SPLINE
SPL {X  -136.861, Y  +292.299, Z    +0.000, E1   +47.815, E3 +153540.728}
SPL {X  -156.420, Y  +335.300, Z    +0.000, E1   +31.885, E3 +153548.517}
SPL {X  -161.293, Y  +358.252, Z    +0.000, E1   +18.542, E3 +153550.234}
SPL {X  -162.687, Y  +373.932, Z    +0.000, E1    +7.306, E3 +153550.370}
SPL {X  -162.820, Y  +382.772, Z    +0.000, E1    -0.135, E3 +153549.808}
SPL {X  -162.820, Y  +387.649, Z    +0.000, E1    -8.215, E3 +153549.563}
SPL {X  -162.820, Y  +392.460, Z    +0.000, E1   -17.627, E3 +153549.544}
SPL {X  -162.820, Y  +397.383, Z    +0.000, E1   -27.100, E3 +153549.614}
SPL {X  -162.820, Y  +404.822, Z    +0.000, E1   -40.113, E3 +153549.266}
SPL {X  -162.820, Y  +416.103, Z    +0.000, E1   -54.033, E3 +153549.118}
SPL {X  -162.820, Y  +467.510, Z    +0.000, E1   -69.867, E3 +153562.696}
SPL {X  -162.820, Y  +604.717, Z    +0.000, E1   -70.047, E3 +153644.416}
ENDSPLINE

SPLINE
SPL {X  -162.820, Y  +602.324, Z    +0.000, E1   -67.733, E3 +153661.865}
ENDSPLINE

SPLINE
SPL {X  -162.820, Y  +616.480, Z    +0.000, E1   -67.752, E3 +153673.895}
SPL {X  -162.820, Y  +636.914, Z    +0.000, E1   -67.842, E3 +153690.588}
SPL {X  -162.820, Y  +651.339, Z    +0.000, E1   -67.768, E3 +153703.257}
SPL {X  -162.820, Y  +663.021, Z    +0.000, E1   -67.764, E3 +153713.302}
SPL {X  -162.642, Y  +681.112, Z    +0.000, E1   -67.812, E3 +153728.453}
SPL {X  -161.154, Y  +696.734, Z    +0.000, E1   -67.591, E3 +153743.450}
SPL {X  -159.690, Y  +705.270, Z    +0.000, E1   -67.348, E3 +153752.558}
SPL {X  -157.320, Y  +715.461, Z    +0.000, E1   -67.133, E3 +153763.151}
SPL {X  -154.452, Y  +725.025, Z    +0.000, E1   -66.701, E3 +153774.335}
SPL {X  -152.159, Y  +731.448, Z    +0.000, E1   -66.356, E3 +153782.288}
SPL {X  -148.374, Y  +740.549, Z    +0.000, E1   -65.919, E3 +153793.162}
SPL {X  -144.196, Y  +749.116, Z    +0.000, E1   -65.203, E3 +153804.838}
SPL {X  -141.115, Y  +754.722, Z    +0.000, E1   -64.893, E3 +153811.297}
SPL {X  -138.151, Y  +759.667, Z    +0.000, E1   -64.251, E3 +153819.119}
SPL {X  -134.751, Y  +764.892, Z    +0.000, E1   -63.716, E3 +153826.122}
SPL {X  -131.007, Y  +770.183, Z    +0.000, E1   -63.497, E3 +153831.619}
SPL {X   -85.750, Y  +811.910, Z    +0.000, E1   -55.921, E3 +153935.572}
ENDSPLINE

SPLINE
SPL {X  -114.463, Y  +789.295, Z    +0.000, E1   -54.865, E3 +154104.839}
SPL {X  -149.148, Y  +738.810, Z    +0.000, E1   -41.467, E3 +154115.910}
SPL {X  -159.693, Y  +705.258, Z    +0.000, E1   -25.118, E3 +154118.550}
SPL {X  -162.196, Y  +687.741, Z    +0.000, E1   -13.310, E3 +154119.515}
SPL {X  -162.791, Y  +676.596, Z    +0.000, E1    -4.586, E3 +154119.799}
SPL {X  -162.820, Y  +671.385, Z    +0.000, E1    +0.078, E3 +154119.216}
SPL {X  -162.820, Y  +667.797, Z    +0.000, E1    +5.943, E3 +154118.875}
SPL {X  -162.820, Y  +663.306, Z    +0.000, E1   +14.820, E3 +154118.842}
SPL {X  -162.820, Y  +658.944, Z    +0.000, E1   +23.544, E3 +154119.031}
SPL {X  -162.820, Y  +650.349, Z    +0.000, E1   +39.427, E3 +154118.528}
SPL {X  -162.820, Y  +632.228, Z    +0.000, E1   +60.508, E3 +154117.758}
SPL {X  -162.820, Y  +572.535, Z    +0.000, E1   +70.270, E3 +154139.803}
SPL {X  -162.820, Y  +446.522, Z    +0.000, E1   +69.253, E3 +154223.626}
SPL {X  -162.820, Y  +444.665, Z    +0.000, E1   +68.107, E3 +154235.177}
SPL {X  -162.820, Y  +425.935, Z    +0.000, E1   +68.194, E3 +154250.232}
SPL {X  -162.820, Y  +409.792, Z    +0.000, E1   +68.121, E3 +154264.156}
SPL {X  -162.820, Y  +394.392, Z    +0.000, E1   +68.165, E3 +154276.730}
SPL {X  -162.820, Y  +385.264, Z    +0.000, E1   +67.766, E3 +154287.646}
ENDSPLINE

SPLINE
SPL {X  -162.820, Y  +401.104, Z    +0.000, E1   +65.023, E3 +154295.371}
ENDSPLINE

SPLINE
SPL {X  -162.820, Y  +386.513, Z    +0.000, E1   +65.423, E3 +154306.367}
SPL {X  -161.886, Y  +363.082, Z    +0.000, E1   +66.474, E3 +154319.799}
SPL {X  -158.043, Y  +341.350, Z    +0.000, E1   +67.216, E3 +154332.995}
SPL {X  -154.848, Y  +330.175, Z    +0.000, E1   +66.891, E3 +154344.807}
SPL {X  -151.242, Y  +320.199, Z    +0.000, E1   +66.443, E3 +154356.608}
SPL {X  -147.540, Y  +311.636, Z    +0.000, E1   +65.718, E3 +154368.586}
SPL {X  -144.094, Y  +304.689, Z    +0.000, E1   +65.338, E3 +154376.801}
SPL {X  -141.093, Y  +299.241, Z    +0.000, E1   +65.039, E3 +154383.114}
SPL {X  -138.425, Y  +294.774, Z    +0.000, E1   +64.416, E3 +154390.297}
SPL {X  -135.581, Y  +290.344, Z    +0.000, E1   +63.996, E3 +154396.130}
SPL {X  -132.317, Y  +285.618, Z    +0.000, E1   +63.461, E3 +154402.704}
SPL {X  -126.028, Y  +277.411, Z    +0.000, E1   +65.004, E3 +154402.876}
SPL {X   -85.291, Y  +241.807, Z    +0.000, E1   +53.957, E3 +154549.471}
ENDSPLINE

SPLINE
SPL {X  -136.861, Y  +292.299, Z    +0.000, E1   +47.815, E3 +154677.091}
SPL {X  -156.420, Y  +335.300, Z    +0.000, E1   +31.885, E3 +154684.881}
SPL {X  -161.293, Y  +358.252, Z    +0.000, E1   +18.542, E3 +154686.598}
SPL {X  -162.487, Y  +370.094, Z    +0.000, E1   +10.144, E3 +154686.676}
SPL {X  -162.818, Y  +379.612, Z    +0.000, E1    +2.663, E3 +154686.652}
SPL {X  -162.820, Y  +382.500, Z    +0.000, E1    +0.000, E3 +154686.245}
SPL {X  -162.820, Y  +383.629, Z    +0.000, E1    -1.565, E3 +154685.939}
SPL {X  -162.820, Y  +387.649, Z    +0.000, E1    -8.215, E3 +154685.926}
SPL {X  -162.820, Y  +392.460, Z    +0.000, E1   -17.627, E3 +154685.908}
SPL {X  -162.820, Y  +397.383, Z    +0.000, E1   -27.100, E3 +154685.978}
SPL {X  -162.820, Y  +404.822, Z    +0.000, E1   -40.113, E3 +154685.630}
SPL {X  -162.820, Y  +416.103, Z    +0.000, E1   -54.033, E3 +154685.482}
SPL {X  -162.820, Y  +472.592, Z    +0.000, E1   -70.190, E3 +154701.084}
SPL {X  -162.820, Y  +605.049, Z    +0.000, E1   -68.347, E3 +154795.565}
SPL {X  -162.820, Y  +616.480, Z    +0.000, E1   -67.752, E3 +154810.258}
SPL {X  -162.820, Y  +631.154, Z    +0.000, E1   -67.735, E3 +154822.793}
SPL {X  -162.820, Y  +647.590, Z    +0.000, E1   -67.861, E3 +154835.828}
SPL {X  -162.820, Y  +663.021, Z    +0.000, E1   -67.764, E3 +154849.666}
SPL {X  -162.642, Y  +681.112, Z    +0.000, E1   -67.812, E3 +154864.817}
SPL {X  -161.154, Y  +696.734, Z    +0.000, E1   -67.591, E3 +154879.814}
SPL {X  -158.503, Y  +710.744, Z    +0.000, E1   -67.284, E3 +154894.345}
SPL {X  -155.060, Y  +723.165, Z    +0.000, E1   -66.797, E3 +154908.521}
SPL {X  -151.511, Y  +733.123, Z    +0.000, E1   -66.286, E3 +154920.675}
SPL {X  -147.735, Y  +741.944, Z    +0.000, E1   -65.827, E3 +154931.201}
SPL {X  -144.196, Y  +749.116, Z    +0.000, E1   -65.203, E3 +154941.201}
SPL {X  -139.960, Y  +756.696, Z    +0.000, E1   -64.606, E3 +154951.096}
SPL {X  -135.604, Y  +763.621, Z    +0.000, E1   -63.883, E3 +154960.698}
SPL {X  -131.007, Y  +770.183, Z    +0.000, E1   -63.497, E3 +154967.983}
SPL {X   -85.750, Y  +811.910, Z    +0.000, E1   -55.921, E3 +155071.935}
ENDSPLINE

SPLINE
SPL {X  -114.463, Y  +789.295, Z    +0.000, E1   -54.865, E3 +155241.202}
SPL {X  -149.148, Y  +738.810, Z    +0.000, E1   -41.467, E3 +155252.274}
SPL {X  -159.693, Y  +705.258, Z    +0.000, E1   -25.118, E3 +155254.913}
SPL {X  -162.196, Y  +687.741, Z    +0.000, E1   -13.310, E3 +155255.878}
SPL {X  -162.791, Y  +676.596, Z    +0.000, E1    -4.586, E3 +155256.163}
SPL {X  -162.820, Y  +671.548, Z    +0.000, E1    -0.068, E3 +155255.640}
SPL {X  -162.820, Y  +669.949, Z    +0.000, E1    +2.213, E3 +155255.327}
SPL {X  -162.820, Y  +664.754, Z    +0.000, E1   +11.697, E3 +155255.226}
SPL {X  -162.820, Y  +658.944, Z    +0.000, E1   +23.544, E3 +155255.394}
SPL {X  -162.820, Y  +653.429, Z    +0.000, E1   +34.521, E3 +155254.785}
SPL {X  -162.820, Y  +647.179, Z    +0.000, E1   +44.317, E3 +155255.001}
SPL {X  -162.820, Y  +632.228, Z    +0.000, E1   +60.508, E3 +155254.121}
SPL {X  -162.820, Y  +572.535, Z    +0.000, E1   +70.270, E3 +155276.166}
SPL {X  -162.820, Y  +446.522, Z    +0.000, E1   +69.253, E3 +155359.990}
SPL {X  -162.820, Y  +444.665, Z    +0.000, E1   +68.107, E3 +155371.540}
SPL {X  -162.820, Y  +425.935, Z    +0.000, E1   +68.194, E3 +155386.596}
SPL {X  -162.820, Y  +405.187, Z    +0.000, E1   +68.161, E3 +155404.184}
SPL {X  -162.820, Y  +387.680, Z    +0.000, E1   +67.977, E3 +155420.373}
ENDSPLINE

SPLINE
SPL {X  -162.820, Y  +397.358, Z    +0.000, E1   +65.083, E3 +155435.011}
ENDSPLINE

SPLINE
SPL {X  -162.719, Y  +374.774, Z    +0.000, E1   +65.968, E3 +155449.496}
SPL {X  -160.017, Y  +350.416, Z    +0.000, E1   +67.091, E3 +155462.401}
SPL {X  -156.713, Y  +336.324, Z    +0.000, E1   +67.030, E3 +155474.998}
SPL {X  -153.279, Y  +325.584, Z    +0.000, E1   +66.662, E3 +155486.763}
SPL {X  -149.546, Y  +316.107, Z    +0.000, E1   +66.216, E3 +155497.938}
SPL {X  -147.033, Y  +310.560, Z    +0.000, E1   +65.497, E3 +155507.153}
SPL {X  -144.094, Y  +304.689, Z    +0.000, E1   +65.338, E3 +155513.164}
SPL {X  -141.093, Y  +299.241, Z    +0.000, E1   +65.039, E3 +155519.477}
SPL {X  -138.425, Y  +294.774, Z    +0.000, E1   +64.416, E3 +155526.661}
SPL {X  -134.374, Y  +288.555, Z    +0.000, E1   +63.758, E3 +155535.303}
SPL {X  -128.896, Y  +281.020, Z    +0.000, E1   +64.005, E3 +155540.426}
SPL {X   -85.291, Y  +241.807, Z    +0.000, E1   +53.957, E3 +155685.834}
ENDSPLINE

SPLINE
SPL {X  -136.861, Y  +292.299, Z    +0.000, E1   +47.815, E3 +155813.455}
SPL {X  -156.420, Y  +335.300, Z    +0.000, E1   +31.885, E3 +155821.244}
SPL {X  -161.293, Y  +358.252, Z    +0.000, E1   +18.542, E3 +155822.962}
SPL {X  -162.487, Y  +370.094, Z    +0.000, E1   +10.144, E3 +155823.040}
SPL {X  -162.818, Y  +379.612, Z    +0.000, E1    +2.663, E3 +155823.015}
SPL {X  -162.820, Y  +382.500, Z    +0.000, E1    +0.000, E3 +155822.609}
SPL {X  -162.820, Y  +383.629, Z    +0.000, E1    -1.565, E3 +155822.302}
SPL {X  -162.820, Y  +387.649, Z    +0.000, E1    -8.215, E3 +155822.290}
SPL {X  -162.820, Y  +392.460, Z    +0.000, E1   -17.627, E3 +155822.271}
SPL {X  -162.820, Y  +397.383, Z    +0.000, E1   -27.100, E3 +155822.342}
SPL {X  -162.820, Y  +404.822, Z    +0.000, E1   -40.113, E3 +155821.993}
SPL {X  -162.820, Y  +416.103, Z    +0.000, E1   -54.033, E3 +155821.845}
SPL {X  -162.820, Y  +467.510, Z    +0.000, E1   -69.867, E3 +155835.423}
SPL {X  -162.820, Y  +604.717, Z    +0.000, E1   -70.047, E3 +155917.143}
ENDSPLINE

SPLINE
SPL {X  -162.820, Y  +602.324, Z    +0.000, E1   -67.733, E3 +155934.592}
ENDSPLINE

SPLINE
SPL {X  -162.820, Y  +616.480, Z    +0.000, E1   -67.752, E3 +155946.622}
SPL {X  -162.820, Y  +636.914, Z    +0.000, E1   -67.842, E3 +155963.316}
SPL {X  -162.820, Y  +654.663, Z    +0.000, E1   -67.744, E3 +155979.142}
SPL {X  -162.820, Y  +673.210, Z    +0.000, E1   -67.837, E3 +155994.175}
SPL {X  -162.071, Y  +689.103, Z    +0.000, E1   -67.763, E3 +156008.240}
SPL {X  -160.373, Y  +701.624, Z    +0.000, E1   -67.439, E3 +156021.599}
SPL {X  -157.887, Y  +713.277, Z    +0.000, E1   -67.197, E3 +156033.370}
SPL {X  -155.060, Y  +723.165, Z    +0.000, E1   -66.797, E3 +156044.885}
SPL {X  -151.511, Y  +733.123, Z    +0.000, E1   -66.286, E3 +156057.039}
SPL {X  -148.440, Y  +740.403, Z    +0.000, E1   -65.944, E3 +156065.399}
SPL {X  -146.076, Y  +745.418, Z    +0.000, E1   -65.453, E3 +156072.874}
SPL {X  -142.207, Y  +752.793, Z    +0.000, E1   -65.028, E3 +156081.723}
SPL {X  -139.223, Y  +757.923, Z    +0.000, E1   -64.359, E3 +156089.693}
SPL {X  -135.604, Y  +763.621, Z    +0.000, E1   -63.883, E3 +156097.061}
SPL {X  -131.007, Y  +770.183, Z    +0.000, E1   -63.497, E3 +156104.346}
SPL {X   -85.750, Y  +811.910, Z    +0.000, E1   -55.921, E3 +156208.299}
ENDSPLINE

SPLINE
SPL {X  -114.463, Y  +789.295, Z    +0.000, E1   -54.865, E3 +156377.566}
SPL {X  -144.553, Y  +748.431, Z    +0.000, E1   -44.979, E3 +156388.274}
SPL {X  -156.024, Y  +720.050, Z    +0.000, E1   -33.178, E3 +156389.841}
SPL {X  -160.714, Y  +699.606, Z    +0.000, E1   -21.520, E3 +156391.715}
SPL {X  -162.196, Y  +687.741, Z    +0.000, E1   -13.310, E3 +156392.242}
SPL {X  -162.718, Y  +679.252, Z    +0.000, E1    -6.705, E3 +156392.579}
SPL {X  -162.820, Y  +671.587, Z    +0.000, E1    -0.252, E3 +156391.978}
SPL {X  -162.820, Y  +667.797, Z    +0.000, E1    +5.943, E3 +156391.602}
SPL {X  -162.820, Y  +663.306, Z    +0.000, E1   +14.820, E3 +156391.569}
SPL {X  -162.820, Y  +658.944, Z    +0.000, E1   +23.544, E3 +156391.758}
SPL {X  -162.820, Y  +650.349, Z    +0.000, E1   +39.427, E3 +156391.255}
SPL {X  -162.820, Y  +635.494, Z    +0.000, E1   +57.613, E3 +156390.958}
SPL {X  -162.820, Y  +626.637, Z    +0.000, E1   +64.941, E3 +156389.674}
SPL {X  -162.820, Y  +572.535, Z    +0.000, E1   +70.270, E3 +156412.530}
SPL {X  -162.820, Y  +446.522, Z    +0.000, E1   +69.253, E3 +156496.354}
SPL {X  -162.820, Y  +444.665, Z    +0.000, E1   +68.107, E3 +156507.904}
SPL {X  -162.820, Y  +425.935, Z    +0.000, E1   +68.194, E3 +156522.960}
SPL {X  -162.820, Y  +409.792, Z    +0.000, E1   +68.121, E3 +156536.883}
SPL {X  -162.820, Y  +394.392, Z    +0.000, E1   +68.165, E3 +156549.458}
SPL {X  -162.820, Y  +385.264, Z    +0.000, E1   +67.766, E3 +156560.373}
ENDSPLINE

SPLINE
SPL {X  -162.820, Y  +401.104, Z    +0.000, E1   +65.023, E3 +156568.098}
ENDSPLINE

SPLINE
SPL {X  -162.820, Y  +386.513, Z    +0.000, E1   +65.423, E3 +156579.094}
SPL {X  -162.431, Y  +369.249, Z    +0.000, E1   +66.195, E3 +156589.095}
SPL {X  -160.017, Y  +350.416, Z    +0.000, E1   +67.091, E3 +156598.765}
SPL {X  -156.713, Y  +336.324, Z    +0.000, E1   +67.030, E3 +156611.361}
SPL {X  -153.279, Y  +325.584, Z    +0.000, E1   +66.662, E3 +156623.126}
SPL {X  -149.546, Y  +316.107, Z    +0.000, E1   +66.216, E3 +156634.302}
SPL {X  -147.033, Y  +310.560, Z    +0.000, E1   +65.497, E3 +156643.516}
SPL {X  -144.094, Y  +304.689, Z    +0.000, E1   +65.338, E3 +156649.528}
SPL {X  -141.093, Y  +299.241, Z    +0.000, E1   +65.039, E3 +156655.841}
SPL {X  -138.425, Y  +294.774, Z    +0.000, E1   +64.416, E3 +156663.025}
SPL {X  -135.581, Y  +290.344, Z    +0.000, E1   +63.996, E3 +156668.857}
SPL {X  -133.378, Y  +287.116, Z    +0.000, E1   +63.482, E3 +156674.021}
SPL {X  -128.896, Y  +281.020, Z    +0.000, E1   +64.005, E3 +156676.790}
SPL {X   -85.291, Y  +241.807, Z    +0.000, E1   +53.957, E3 +156822.198}
ENDSPLINE

SPLINE
SPL {X  -136.861, Y  +292.299, Z    +0.000, E1   +47.815, E3 +156949.819}
SPL {X  -156.420, Y  +335.300, Z    +0.000, E1   +31.885, E3 +156957.608}
SPL {X  -161.293, Y  +358.252, Z    +0.000, E1   +18.542, E3 +156959.325}
SPL {X  -162.487, Y  +370.094, Z    +0.000, E1   +10.144, E3 +156959.404}
SPL {X  -162.818, Y  +379.612, Z    +0.000, E1    +2.663, E3 +156959.379}
SPL {X  -162.820, Y  +382.928, Z    +0.000, E1    -0.395, E3 +156958.856}
SPL {X  -162.820, Y  +386.448, Z    +0.000, E1    -6.246, E3 +156958.611}
SPL {X  -162.820, Y  +391.031, Z    +0.000, E1   -14.627, E3 +156958.670}
SPL {X  -162.820, Y  +397.383, Z    +0.000, E1   -27.100, E3 +156958.705}
SPL {X  -162.820, Y  +404.822, Z    +0.000, E1   -40.113, E3 +156958.357}
SPL {X  -162.820, Y  +416.103, Z    +0.000, E1   -54.033, E3 +156958.209}
SPL {X  -162.820, Y  +467.510, Z    +0.000, E1   -69.867, E3 +156971.787}
SPL {X  -162.820, Y  +604.717, Z    +0.000, E1   -70.047, E3 +157053.507}
SPL {X  -162.820, Y  +606.663, Z    +0.000, E1   -67.762, E3 +157074.555}
SPL {X  -162.820, Y  +620.455, Z    +0.000, E1   -67.717, E3 +157086.528}
SPL {X  -162.820, Y  +636.914, Z    +0.000, E1   -67.842, E3 +157099.679}
SPL {X  -162.820, Y  +654.663, Z    +0.000, E1   -67.744, E3 +157115.505}
SPL {X  -162.820, Y  +673.210, Z    +0.000, E1   -67.837, E3 +157130.539}
SPL {X  -162.071, Y  +689.103, Z    +0.000, E1   -67.763, E3 +157144.604}
SPL {X  -160.908, Y  +698.381, Z    +0.000, E1   -67.466, E3 +157154.843}
SPL {X  -159.690, Y  +705.270, Z    +0.000, E1   -67.348, E3 +157161.648}
SPL {X  -157.320, Y  +715.461, Z    +0.000, E1   -67.133, E3 +157172.242}
SPL {X  -154.452, Y  +725.025, Z    +0.000, E1   -66.701, E3 +157183.426}
SPL {X  -151.511, Y  +733.123, Z    +0.000, E1   -66.286, E3 +157193.402}
SPL {X  -147.735, Y  +741.944, Z    +0.000, E1   -65.827, E3 +157203.928}
SPL {X  -144.196, Y  +749.116, Z    +0.000, E1   -65.203, E3 +157213.929}
SPL {X  -139.960, Y  +756.696, Z    +0.000, E1   -64.606, E3 +157223.823}
SPL {X  -136.860, Y  +761.702, Z    +0.000, E1   -64.057, E3 +157230.817}
SPL {X  -134.751, Y  +764.892, Z    +0.000, E1   -63.716, E3 +157235.212}
SPL {X  -131.007, Y  +770.183, Z    +0.000, E1   -63.497, E3 +157240.710}
SPL {X   -85.750, Y  +811.910, Z    +0.000, E1   -55.921, E3 +157344.663}
ENDSPLINE

SPLINE
SPL {X  -114.463, Y  +789.295, Z    +0.000, E1   -54.865, E3 +157513.930}
SPL {X  -149.148, Y  +738.810, Z    +0.000, E1   -41.467, E3 +157525.001}
SPL {X  -159.693, Y  +705.258, Z    +0.000, E1   -25.118, E3 +157527.640}
SPL {X  -162.196, Y  +687.741, Z    +0.000, E1   -13.310, E3 +157528.606}
SPL {X  -162.718, Y  +679.252, Z    +0.000, E1    -6.705, E3 +157528.943}
SPL {X  -162.820, Y  +671.809, Z    +0.000, E1    -0.439, E3 +157528.409}
SPL {X  -162.820, Y  +669.949, Z    +0.000, E1    +2.213, E3 +157528.054}
SPL {X  -162.820, Y  +664.754, Z    +0.000, E1   +11.697, E3 +157527.953}
SPL {X  -162.820, Y  +658.944, Z    +0.000, E1   +23.544, E3 +157528.122}
SPL {X  -162.820, Y  +650.349, Z    +0.000, E1   +39.427, E3 +157527.619}
SPL {X  -162.820, Y  +632.228, Z    +0.000, E1   +60.508, E3 +157526.849}
SPL {X  -162.820, Y  +572.535, Z    +0.000, E1   +70.270, E3 +157548.893}
SPL {X  -162.820, Y  +446.522, Z    +0.000, E1   +69.253, E3 +157632.717}
SPL {X  -162.820, Y  +444.665, Z    +0.000, E1   +68.107, E3 +157644.267}
SPL {X  -162.820, Y  +425.935, Z    +0.000, E1   +68.194, E3 +157659.323}
SPL {X  -162.820, Y  +405.187, Z    +0.000, E1   +68.161, E3 +157676.912}
SPL {X  -162.820, Y  +387.680, Z    +0.000, E1   +67.977, E3 +157693.100}
ENDSPLINE

SPLINE
SPL {X  -162.820, Y  +397.358, Z    +0.000, E1   +65.083, E3 +157707.739}
ENDSPLINE

SPLINE
SPL {X  -162.719, Y  +374.774, Z    +0.000, E1   +65.968, E3 +157722.223}
SPL {X  -160.017, Y  +350.416, Z    +0.000, E1   +67.091, E3 +157735.129}
SPL {X  -156.713, Y  +336.324, Z    +0.000, E1   +67.030, E3 +157747.725}
SPL {X  -153.279, Y  +325.584, Z    +0.000, E1   +66.662, E3 +157759.490}
SPL {X  -150.291, Y  +317.867, Z    +0.000, E1   +66.312, E3 +157768.409}
SPL {X  -147.540, Y  +311.636, Z    +0.000, E1   +65.718, E3 +157777.677}
SPL {X  -144.094, Y  +304.689, Z    +0.000, E1   +65.338, E3 +157785.892}
SPL {X  -141.093, Y  +299.241, Z    +0.000, E1   +65.039, E3 +157792.204}
SPL {X  -138.425, Y  +294.774, Z    +0.000, E1   +64.416, E3 +157799.388}
SPL {X  -134.374, Y  +288.555, Z    +0.000, E1   +63.758, E3 +157808.031}
SPL {X  -128.896, Y  +281.020, Z    +0.000, E1   +64.005, E3 +157813.153}
SPL {X   -85.291, Y  +241.807, Z    +0.000, E1   +53.957, E3 +157958.561}
ENDSPLINE

SPLINE
SPL {X  -136.861, Y  +292.299, Z    +0.000, E1   +47.815, E3 +158086.182}
SPL {X  -156.420, Y  +335.300, Z    +0.000, E1   +31.885, E3 +158093.972}
SPL {X  -161.293, Y  +358.252, Z    +0.000, E1   +18.542, E3 +158095.689}
SPL {X  -162.487, Y  +370.094, Z    +0.000, E1   +10.144, E3 +158095.767}
SPL {X  -162.818, Y  +379.612, Z    +0.000, E1    +2.663, E3 +158095.743}
SPL {X  -162.820, Y  +382.928, Z    +0.000, E1    -0.395, E3 +158095.220}
SPL {X  -162.820, Y  +387.649, Z    +0.000, E1    -8.215, E3 +158095.017}
SPL {X  -162.820, Y  +392.460, Z    +0.000, E1   -17.627, E3 +158094.999}
SPL {X  -162.820, Y  +397.383, Z    +0.000, E1   -27.100, E3 +158095.069}
SPL {X  -162.820, Y  +404.822, Z    +0.000, E1   -40.113, E3 +158094.720}
SPL {X  -162.820, Y  +416.103, Z    +0.000, E1   -54.033, E3 +158094.573}
SPL {X  -162.820, Y  +472.592, Z    +0.000, E1   -70.190, E3 +158110.175}
SPL {X  -162.820, Y  +611.623, Z    +0.000, E1   -69.722, E3 +158197.507}
ENDSPLINE

SPLINE
SPL {X  -162.820, Y  +606.663, Z    +0.000, E1   -67.762, E3 +158210.919}
ENDSPLINE

SPLINE
SPL {X  -162.820, Y  +626.641, Z    +0.000, E1   -67.759, E3 +158228.026}
SPL {X  -162.820, Y  +643.417, Z    +0.000, E1   -67.904, E3 +158240.843}
SPL {X  -162.820, Y  +654.663, Z    +0.000, E1   -67.744, E3 +158251.869}
SPL {X  -162.820, Y  +673.210, Z    +0.000, E1   -67.837, E3 +158266.902}
SPL {X  -162.338, Y  +686.018, Z    +0.000, E1   -67.736, E3 +158278.484}
SPL {X  -161.154, Y  +696.734, Z    +0.000, E1   -67.591, E3 +158288.905}
SPL {X  -159.690, Y  +705.270, Z    +0.000, E1   -67.348, E3 +158298.012}
SPL {X  -157.887, Y  +713.277, Z    +0.000, E1   -67.197, E3 +158306.098}
SPL {X  -155.060, Y  +723.165, Z    +0.000, E1   -66.797, E3 +158317.612}
SPL {X  -152.159, Y  +731.448, Z    +0.000, E1   -66.356, E3 +158327.743}
SPL {X  -149.129, Y  +738.853, Z    +0.000, E1   -66.010, E3 +158336.440}
SPL {X  -146.076, Y  +745.418, Z    +0.000, E1   -65.453, E3 +158345.602}
SPL {X  -143.238, Y  +750.916, Z    +0.000, E1   -65.112, E3 +158352.286}
SPL {X  -139.960, Y  +756.696, Z    +0.000, E1   -64.606, E3 +158360.187}
SPL {X  -136.860, Y  +761.702, Z    +0.000, E1   -64.057, E3 +158367.181}
SPL {X  -134.751, Y  +764.892, Z    +0.000, E1   -63.716, E3 +158371.576}
SPL {X  -131.007, Y  +770.183, Z    +0.000, E1   -63.497, E3 +158377.074}
SPL {X   -85.750, Y  +811.910, Z    +0.000, E1   -55.921, E3 +158481.026}
ENDSPLINE

SPLINE
SPL {X  -114.463, Y  +789.295, Z    +0.000, E1   -54.865, E3 +158650.293}
SPL {X  -149.148, Y  +738.810, Z    +0.000, E1   -41.467, E3 +158661.364}
SPL {X  -159.693, Y  +705.258, Z    +0.000, E1   -25.118, E3 +158664.004}
SPL {X  -162.196, Y  +687.741, Z    +0.000, E1   -13.310, E3 +158664.969}
SPL {X  -162.791, Y  +676.596, Z    +0.000, E1    -4.586, E3 +158665.253}
SPL {X  -162.820, Y  +671.548, Z    +0.000, E1    -0.068, E3 +158664.730}
SPL {X  -162.820, Y  +669.949, Z    +0.000, E1    +2.213, E3 +158664.418}
SPL {X  -162.820, Y  +664.754, Z    +0.000, E1   +11.697, E3 +158664.317}
SPL {X  -162.820, Y  +658.944, Z    +0.000, E1   +23.544, E3 +158664.485}
SPL {X  -162.820, Y  +653.429, Z    +0.000, E1   +34.521, E3 +158663.876}
SPL {X  -162.820, Y  +647.179, Z    +0.000, E1   +44.317, E3 +158664.092}
SPL {X  -162.820, Y  +632.228, Z    +0.000, E1   +60.508, E3 +158663.212}
SPL {X  -162.820, Y  +572.535, Z    +0.000, E1   +70.270, E3 +158685.257}
SPL {X  -162.820, Y  +446.522, Z    +0.000, E1   +69.253, E3 +158769.081}
SPL {X  -162.820, Y  +440.686, Z    +0.000, E1   +68.127, E3 +158783.956}
SPL {X  -162.820, Y  +421.575, Z    +0.000, E1   +68.212, E3 +158799.019}
SPL {X  -162.820, Y  +409.792, Z    +0.000, E1   +68.121, E3 +158809.611}
SPL {X  -162.820, Y  +394.392, Z    +0.000, E1   +68.165, E3 +158822.185}
SPL {X  -162.820, Y  +385.264, Z    +0.000, E1   +67.766, E3 +158833.100}
ENDSPLINE

SPLINE
SPL {X  -162.820, Y  +401.104, Z    +0.000, E1   +65.023, E3 +158840.826}
ENDSPLINE

SPLINE
SPL {X  -162.820, Y  +386.513, Z    +0.000, E1   +65.423, E3 +158851.821}
SPL {X  -161.886, Y  +363.082, Z    +0.000, E1   +66.474, E3 +158865.254}
SPL {X  -158.765, Y  +344.387, Z    +0.000, E1   +67.403, E3 +158874.155}
SPL {X  -157.549, Y  +339.407, Z    +0.000, E1   +67.028, E3 +158881.368}
SPL {X  -154.848, Y  +330.175, Z    +0.000, E1   +66.891, E3 +158890.261}
SPL {X  -152.657, Y  +323.878, Z    +0.000, E1   +66.551, E3 +158897.996}
SPL {X  -149.546, Y  +316.107, Z    +0.000, E1   +66.216, E3 +158907.029}
SPL {X  -147.033, Y  +310.560, Z    +0.000, E1   +65.497, E3 +158916.244}
SPL {X  -144.094, Y  +304.689, Z    +0.000, E1   +65.338, E3 +158922.255}
SPL {X  -141.093, Y  +299.241, Z    +0.000, E1   +65.039, E3 +158928.568}
SPL {X  -138.425, Y  +294.774, Z    +0.000, E1   +64.416, E3 +158935.752}
SPL {X  -134.374, Y  +288.555, Z    +0.000, E1   +63.758, E3 +158944.394}
SPL {X  -128.896, Y  +281.020, Z    +0.000, E1   +64.005, E3 +158949.517}
SPL {X   -85.291, Y  +241.807, Z    +0.000, E1   +53.957, E3 +159094.925}
ENDSPLINE

SPLINE
SPL {X  -136.861, Y  +292.299, Z    +0.000, E1   +47.815, E3 +159222.546}
SPL {X  -156.420, Y  +335.300, Z    +0.000, E1   +31.885, E3 +159230.335}
SPL {X  -161.293, Y  +358.252, Z    +0.000, E1   +18.542, E3 +159232.053}
SPL {X  -162.487, Y  +370.094, Z    +0.000, E1   +10.144, E3 +159232.131}
SPL {X  -162.818, Y  +379.612, Z    +0.000, E1    +2.663, E3 +159232.106}
SPL {X  -162.820, Y  +382.928, Z    +0.000, E1    -0.395, E3 +159231.584}
SPL {X  -162.820, Y  +387.649, Z    +0.000, E1    -8.215, E3 +159231.381}
SPL {X  -162.820, Y  +392.460, Z    +0.000, E1   -17.627, E3 +159231.362}
SPL {X  -162.820, Y  +397.383, Z    +0.000, E1   -27.100, E3 +159231.433}
SPL {X  -162.820, Y  +404.822, Z    +0.000, E1   -40.113, E3 +159231.084}
SPL {X  -162.820, Y  +416.103, Z    +0.000, E1   -54.033, E3 +159230.936}
SPL {X  -162.820, Y  +467.510, Z    +0.000, E1   -69.867, E3 +159244.514}
SPL {X  -162.820, Y  +604.717, Z    +0.000, E1   -70.047, E3 +159326.234}
ENDSPLINE

SPLINE
SPL {X  -162.820, Y  +602.324, Z    +0.000, E1   -67.733, E3 +159343.683}
ENDSPLINE

SPLINE
SPL {X  -162.820, Y  +616.480, Z    +0.000, E1   -67.752, E3 +159355.713}
SPL {X  -162.820, Y  +636.914, Z    +0.000, E1   -67.842, E3 +159372.407}
SPL {X  -162.820, Y  +654.663, Z    +0.000, E1   -67.744, E3 +159388.233}
SPL {X  -162.820, Y  +673.210, Z    +0.000, E1   -67.837, E3 +159403.266}
SPL {X  -162.071, Y  +689.103, Z    +0.000, E1   -67.763, E3 +159417.331}
SPL {X  -160.373, Y  +701.624, Z    +0.000, E1   -67.439, E3 +159430.690}
SPL {X  -157.887, Y  +713.277, Z    +0.000, E1   -67.197, E3 +159442.461}
SPL {X  -155.060, Y  +723.165, Z    +0.000, E1   -66.797, E3 +159453.976}
SPL {X  -151.511, Y  +733.123, Z    +0.000, E1   -66.286, E3 +159466.130}
SPL {X  -148.440, Y  +740.403, Z    +0.000, E1   -65.944, E3 +159474.490}
SPL {X  -146.076, Y  +745.418, Z    +0.000, E1   -65.453, E3 +159481.965}
SPL {X  -142.207, Y  +752.793, Z    +0.000, E1   -65.028, E3 +159490.814}
SPL {X  -138.151, Y  +759.667, Z    +0.000, E1   -64.251, E3 +159500.937}
SPL {X  -134.751, Y  +764.892, Z    +0.000, E1   -63.716, E3 +159507.940}
SPL {X  -131.007, Y  +770.183, Z    +0.000, E1   -63.497, E3 +159513.437}
SPL {X   -85.750, Y  +811.910, Z    +0.000, E1   -55.921, E3 +159617.390}
ENDSPLINE

SPLINE
SPL {X  -114.463, Y  +789.295, Z    +0.000, E1   -54.865, E3 +159786.657}
SPL {X  -149.148, Y  +738.810, Z    +0.000, E1   -41.467, E3 +159797.728}
SPL {X  -159.693, Y  +705.258, Z    +0.000, E1   -25.118, E3 +159800.368}
SPL {X  -162.196, Y  +687.741, Z    +0.000, E1   -13.310, E3 +159801.333}
SPL {X  -162.718, Y  +679.252, Z    +0.000, E1    -6.705, E3 +159801.670}
SPL {X  -162.820, Y  +671.587, Z    +0.000, E1    -0.252, E3 +159801.069}
SPL {X  -162.820, Y  +668.947, Z    +0.000, E1    +4.071, E3 +159800.682}
SPL {X  -162.820, Y  +664.754, Z    +0.000, E1   +11.697, E3 +159800.681}
SPL {X  -162.820, Y  +658.944, Z    +0.000, E1   +23.544, E3 +159800.849}
SPL {X  -162.820, Y  +653.429, Z    +0.000, E1   +34.521, E3 +159800.239}
SPL {X  -162.820, Y  +647.179, Z    +0.000, E1   +44.317, E3 +159800.456}
SPL {X  -162.820, Y  +632.228, Z    +0.000, E1   +60.508, E3 +159799.576}
SPL {X  -162.820, Y  +572.535, Z    +0.000, E1   +70.270, E3 +159821.621}
SPL {X  -162.820, Y  +446.522, Z    +0.000, E1   +69.253, E3 +159905.445}
SPL {X  -162.820, Y  +440.686, Z    +0.000, E1   +68.127, E3 +159920.319}
SPL {X  -162.820, Y  +421.575, Z    +0.000, E1   +68.212, E3 +159935.383}
SPL {X  -162.820, Y  +409.792, Z    +0.000, E1   +68.121, E3 +159945.974}
SPL {X  -162.820, Y  +394.392, Z    +0.000, E1   +68.165, E3 +159958.549}
SPL {X  -162.820, Y  +385.264, Z    +0.000, E1   +67.766, E3 +159969.464}
ENDSPLINE

SPLINE
SPL {X  -162.820, Y  +401.104, Z    +0.000, E1   +65.023, E3 +159977.189}
ENDSPLINE

SPLINE
SPL {X  -162.820, Y  +386.513, Z    +0.000, E1   +65.423, E3 +159988.185}
SPL {X  -161.886, Y  +363.082, Z    +0.000, E1   +66.474, E3 +160001.617}
SPL {X  -158.765, Y  +344.387, Z    +0.000, E1   +67.403, E3 +160010.518}
SPL {X  -157.549, Y  +339.407, Z    +0.000, E1   +67.028, E3 +160017.732}
SPL {X  -154.848, Y  +330.175, Z    +0.000, E1   +66.891, E3 +160026.625}
SPL {X  -151.242, Y  +320.199, Z    +0.000, E1   +66.443, E3 +160038.426}
SPL {X  -147.540, Y  +311.636, Z    +0.000, E1   +65.718, E3 +160050.404}
SPL {X  -144.094, Y  +304.689, Z    +0.000, E1   +65.338, E3 +160058.619}
SPL {X  -141.093, Y  +299.241, Z    +0.000, E1   +65.039, E3 +160064.932}
SPL {X  -138.425, Y  +294.774, Z    +0.000, E1   +64.416, E3 +160072.116}
SPL {X  -134.374, Y  +288.555, Z    +0.000, E1   +63.758, E3 +160080.758}
SPL {X  -128.896, Y  +281.020, Z    +0.000, E1   +64.005, E3 +160085.881}
SPL {X   -85.291, Y  +241.807, Z    +0.000, E1   +53.957, E3 +160231.289}
ENDSPLINE

SPLINE
SPL {X  -136.861, Y  +292.299, Z    +0.000, E1   +47.815, E3 +160358.910}
SPL {X  -156.420, Y  +335.300, Z    +0.000, E1   +31.885, E3 +160366.699}
SPL {X  -161.293, Y  +358.252, Z    +0.000, E1   +18.542, E3 +160368.416}
SPL {X  -162.487, Y  +370.094, Z    +0.000, E1   +10.144, E3 +160368.494}
SPL {X  -162.818, Y  +379.612, Z    +0.000, E1    +2.663, E3 +160368.470}
SPL {X  -162.820, Y  +382.500, Z    +0.000, E1    +0.000, E3 +160368.064}
SPL {X  -162.820, Y  +383.629, Z    +0.000, E1    -1.565, E3 +160367.757}
SPL {X  -162.820, Y  +387.649, Z    +0.000, E1    -8.215, E3 +160367.745}
SPL {X  -162.820, Y  +392.460, Z    +0.000, E1   -17.627, E3 +160367.726}
SPL {X  -162.820, Y  +397.383, Z    +0.000, E1   -27.100, E3 +160367.796}
SPL {X  -162.820, Y  +404.822, Z    +0.000, E1   -40.113, E3 +160367.448}
SPL {X  -162.820, Y  +416.103, Z    +0.000, E1   -54.033, E3 +160367.300}
SPL {X  -162.820, Y  +472.592, Z    +0.000, E1   -70.190, E3 +160382.902}
SPL {X  -162.820, Y  +605.049, Z    +0.000, E1   -68.347, E3 +160477.384}
SPL {X  -162.820, Y  +616.480, Z    +0.000, E1   -67.752, E3 +160492.076}
SPL {X  -162.820, Y  +631.154, Z    +0.000, E1   -67.735, E3 +160504.611}
SPL {X  -162.820, Y  +647.590, Z    +0.000, E1   -67.861, E3 +160517.646}
SPL {X  -162.820, Y  +663.021, Z    +0.000, E1   -67.764, E3 +160531.484}
SPL {X  -162.642, Y  +681.112, Z    +0.000, E1   -67.812, E3 +160546.635}
SPL {X  -161.154, Y  +696.734, Z    +0.000, E1   -67.591, E3 +160561.632}
SPL {X  -158.503, Y  +710.744, Z    +0.000, E1   -67.284, E3 +160576.163}
SPL {X  -155.060, Y  +723.165, Z    +0.000, E1   -66.797, E3 +160590.339}
SPL {X  -151.511, Y  +733.123, Z    +0.000, E1   -66.286, E3 +160602.493}
SPL {X  -148.440, Y  +740.403, Z    +0.000, E1   -65.944, E3 +160610.854}
SPL {X  -146.076, Y  +745.418, Z    +0.000, E1   -65.453, E3 +160618.329}
SPL {X  -142.207, Y  +752.793, Z    +0.000, E1   -65.028, E3 +160627.178}
SPL {X  -138.151, Y  +759.667, Z    +0.000, E1   -64.251, E3 +160637.301}
SPL {X  -134.751, Y  +764.892, Z    +0.000, E1   -63.716, E3 +160644.303}
SPL {X  -131.007, Y  +770.183, Z    +0.000, E1   -63.497, E3 +160649.801}
SPL {X   -85.750, Y  +811.910, Z    +0.000, E1   -55.921, E3 +160753.754}
ENDSPLINE

SPLINE
SPL {X  -114.463, Y  +789.295, Z    +0.000, E1   -54.865, E3 +160923.021}
SPL {X  -149.148, Y  +738.810, Z    +0.000, E1   -41.467, E3 +160934.092}
SPL {X  -159.693, Y  +705.258, Z    +0.000, E1   -25.118, E3 +160936.731}
SPL {X  -162.196, Y  +687.741, Z    +0.000, E1   -13.310, E3 +160937.697}
SPL {X  -162.791, Y  +676.596, Z    +0.000, E1    -4.586, E3 +160937.981}
SPL {X  -162.820, Y  +671.548, Z    +0.000, E1    -0.068, E3 +160937.458}
SPL {X  -162.820, Y  +669.949, Z    +0.000, E1    +2.213, E3 +160937.145}
SPL {X  -162.820, Y  +664.754, Z    +0.000, E1   +11.697, E3 +160937.044}
SPL {X  -162.820, Y  +658.944, Z    +0.000, E1   +23.544, E3 +160937.212}
SPL {X  -162.820, Y  +650.349, Z    +0.000, E1   +39.427, E3 +160936.710}
SPL {X  -162.820, Y  +632.228, Z    +0.000, E1   +60.508, E3 +160935.940}
SPL {X  -162.820, Y  +572.535, Z    +0.000, E1   +70.270, E3 +160957.984}
SPL {X  -162.820, Y  +446.522, Z    +0.000, E1   +69.253, E3 +161041.808}
SPL {X  -162.820, Y  +440.686, Z    +0.000, E1   +68.127, E3 +161056.683}
SPL {X  -162.820, Y  +421.575, Z    +0.000, E1   +68.212, E3 +161071.747}
SPL {X  -162.820, Y  +409.792, Z    +0.000, E1   +68.121, E3 +161082.338}
SPL {X  -162.820, Y  +394.392, Z    +0.000, E1   +68.165, E3 +161094.912}
SPL {X  -162.820, Y  +385.264, Z    +0.000, E1   +67.766, E3 +161105.827}
ENDSPLINE

SPLINE
SPL {X  -162.820, Y  +397.358, Z    +0.000, E1   +65.083, E3 +161116.830}
ENDSPLINE

SPLINE
SPL {X  -162.719, Y  +374.774, Z    +0.000, E1   +65.968, E3 +161131.314}
SPL {X  -161.214, Y  +357.685, Z    +0.000, E1   +66.686, E3 +161141.068}
SPL {X  -158.043, Y  +341.350, Z    +0.000, E1   +67.216, E3 +161151.177}
SPL {X  -154.848, Y  +330.175, Z    +0.000, E1   +66.891, E3 +161162.989}
SPL {X  -152.657, Y  +323.878, Z    +0.000, E1   +66.551, E3 +161170.723}
SPL {X  -150.291, Y  +317.867, Z    +0.000, E1   +66.312, E3 +161177.500}
SPL {X  -147.540, Y  +311.636, Z    +0.000, E1   +65.718, E3 +161186.768}
SPL {X  -144.094, Y  +304.689, Z    +0.000, E1   +65.338, E3 +161194.983}
SPL {X  -141.093, Y  +299.241, Z    +0.000, E1   +65.039, E3 +161201.295}
SPL {X  -138.425, Y  +294.774, Z    +0.000, E1   +64.416, E3 +161208.479}
SPL {X  -135.581, Y  +290.344, Z    +0.000, E1   +63.996, E3 +161214.312}
SPL {X  -133.378, Y  +287.116, Z    +0.000, E1   +63.482, E3 +161219.476}
SPL {X  -128.896, Y  +281.020, Z    +0.000, E1   +64.005, E3 +161222.244}
SPL {X   -85.291, Y  +241.807, Z    +0.000, E1   +53.957, E3 +161367.652}
ENDSPLINE

SPLINE
SPL {X  -136.861, Y  +292.299, Z    +0.000, E1   +47.815, E3 +161495.273}
SPL {X  -156.420, Y  +335.300, Z    +0.000, E1   +31.885, E3 +161503.062}
SPL {X  -161.293, Y  +358.252, Z    +0.000, E1   +18.542, E3 +161504.780}
SPL {X  -162.687, Y  +373.932, Z    +0.000, E1    +7.306, E3 +161504.916}
SPL {X  -162.820, Y  +382.772, Z    +0.000, E1    -0.135, E3 +161504.353}
SPL {X  -162.820, Y  +387.649, Z    +0.000, E1    -8.215, E3 +161504.108}
SPL {X  -162.820, Y  +392.460, Z    +0.000, E1   -17.627, E3 +161504.090}
SPL {X  -162.820, Y  +397.383, Z    +0.000, E1   -27.100, E3 +161504.160}
SPL {X  -162.820, Y  +404.822, Z    +0.000, E1   -40.113, E3 +161503.811}
SPL {X  -162.820, Y  +416.103, Z    +0.000, E1   -54.033, E3 +161503.663}
SPL {X  -162.820, Y  +467.510, Z    +0.000, E1   -69.867, E3 +161517.242}
SPL {X  -162.820, Y  +604.717, Z    +0.000, E1   -70.047, E3 +161598.961}
ENDSPLINE

SPLINE
SPL {X  -162.820, Y  +602.324, Z    +0.000, E1   -67.733, E3 +161616.410}
ENDSPLINE

SPLINE
SPL {X  -162.820, Y  +616.480, Z    +0.000, E1   -67.752, E3 +161628.440}
SPL {X  -162.820, Y  +636.914, Z    +0.000, E1   -67.842, E3 +161645.134}
SPL {X  -162.820, Y  +651.339, Z    +0.000, E1   -67.768, E3 +161657.803}
SPL {X  -162.820, Y  +663.021, Z    +0.000, E1   -67.764, E3 +161667.847}
SPL {X  -162.642, Y  +681.112, Z    +0.000, E1   -67.812, E3 +161682.999}
SPL {X  -161.154, Y  +696.734, Z    +0.000, E1   -67.591, E3 +161697.996}
SPL {X  -159.690, Y  +705.270, Z    +0.000, E1   -67.348, E3 +161707.103}
SPL {X  -157.320, Y  +715.461, Z    +0.000, E1   -67.133, E3 +161717.696}
SPL {X  -154.452, Y  +725.025, Z    +0.000, E1   -66.701, E3 +161728.881}
SPL {X  -152.159, Y  +731.448, Z    +0.000, E1   -66.356, E3 +161736.834}
SPL {X  -148.374, Y  +740.549, Z    +0.000, E1   -65.919, E3 +161747.708}
SPL {X  -144.196, Y  +749.116, Z    +0.000, E1   -65.203, E3 +161759.383}
SPL {X  -141.115, Y  +754.722, Z    +0.000, E1   -64.893, E3 +161765.842}
SPL {X  -138.151, Y  +759.667, Z    +0.000, E1   -64.251, E3 +161773.664}
SPL {X  -134.751, Y  +764.892, Z    +0.000, E1   -63.716, E3 +161780.667}
SPL {X  -131.007, Y  +770.183, Z    +0.000, E1   -63.497, E3 +161786.165}
SPL {X   -85.750, Y  +811.910, Z    +0.000, E1   -55.921, E3 +161890.117}
ENDSPLINE

SPLINE
SPL {X  -114.463, Y  +789.295, Z    +0.000, E1   -54.865, E3 +162059.384}
SPL {X  -149.148, Y  +738.810, Z    +0.000, E1   -41.467, E3 +162070.455}
SPL {X  -159.693, Y  +705.258, Z    +0.000, E1   -25.118, E3 +162073.095}
SPL {X  -162.196, Y  +687.741, Z    +0.000, E1   -13.310, E3 +162074.060}
SPL {X  -162.791, Y  +676.596, Z    +0.000, E1    -4.586, E3 +162074.344}
SPL {X  -162.820, Y  +671.385, Z    +0.000, E1    +0.078, E3 +162073.762}
SPL {X  -162.820, Y  +667.797, Z    +0.000, E1    +5.943, E3 +162073.420}
SPL {X  -162.820, Y  +663.306, Z    +0.000, E1   +14.820, E3 +162073.387}
SPL {X  -162.820, Y  +658.944, Z    +0.000, E1   +23.544, E3 +162073.576}
SPL {X  -162.820, Y  +650.349, Z    +0.000, E1   +39.427, E3 +162073.073}
SPL {X  -162.820, Y  +632.228, Z    +0.000, E1   +60.508, E3 +162072.303}
SPL {X  -162.820, Y  +572.535, Z    +0.000, E1   +70.270, E3 +162094.348}
SPL {X  -162.820, Y  +446.522, Z    +0.000, E1   +69.253, E3 +162178.172}
SPL {X  -162.820, Y  +444.665, Z    +0.000, E1   +68.107, E3 +162189.722}
SPL {X  -162.820, Y  +425.935, Z    +0.000, E1   +68.194, E3 +162204.778}
SPL {X  -162.820, Y  +409.792, Z    +0.000, E1   +68.121, E3 +162218.702}
SPL {X  -162.820, Y  +394.392, Z    +0.000, E1   +68.165, E3 +162231.276}
SPL {X  -162.820, Y  +385.264, Z    +0.000, E1   +67.766, E3 +162242.191}
ENDSPLINE

SPLINE
SPL {X  -162.820, Y  +401.104, Z    +0.000, E1   +65.023, E3 +162249.917}
ENDSPLINE

SPLINE
SPL {X  -162.820, Y  +386.513, Z    +0.000, E1   +65.423, E3 +162260.912}
SPL {X  -161.886, Y  +363.082, Z    +0.000, E1   +66.474, E3 +162274.345}
SPL {X  -158.043, Y  +341.350, Z    +0.000, E1   +67.216, E3 +162287.541}
SPL {X  -154.848, Y  +330.175, Z    +0.000, E1   +66.891, E3 +162299.352}
SPL {X  -151.242, Y  +320.199, Z    +0.000, E1   +66.443, E3 +162311.153}
SPL {X  -147.540, Y  +311.636, Z    +0.000, E1   +65.718, E3 +162323.132}
SPL {X  -144.094, Y  +304.689, Z    +0.000, E1   +65.338, E3 +162331.346}
SPL {X  -141.093, Y  +299.241, Z    +0.000, E1   +65.039, E3 +162337.659}
SPL {X  -138.425, Y  +294.774, Z    +0.000, E1   +64.416, E3 +162344.843}
SPL {X  -135.581, Y  +290.344, Z    +0.000, E1   +63.996, E3 +162350.675}
SPL {X  -132.317, Y  +285.618, Z    +0.000, E1   +63.461, E3 +162357.250}
SPL {X  -126.028, Y  +277.411, Z    +0.000, E1   +65.004, E3 +162357.422}
SPL {X   -85.291, Y  +241.807, Z    +0.000, E1   +53.957, E3 +162504.016}
ENDSPLINE

SPLINE
SPL {X  -136.861, Y  +292.299, Z    +0.000, E1   +47.815, E3 +162631.637}
SPL {X  -156.420, Y  +335.300, Z    +0.000, E1   +31.885, E3 +162639.426}
SPL {X  -161.293, Y  +358.252, Z    +0.000, E1   +18.542, E3 +162641.144}
SPL {X  -162.487, Y  +370.094, Z    +0.000, E1   +10.144, E3 +162641.222}
SPL {X  -162.818, Y  +379.612, Z    +0.000, E1    +2.663, E3 +162641.197}
SPL {X  -162.820, Y  +382.500, Z    +0.000, E1    +0.000, E3 +162640.791}
SPL {X  -162.820, Y  +383.629, Z    +0.000, E1    -1.565, E3 +162640.484}
SPL {X  -162.820, Y  +387.649, Z    +0.000, E1    -8.215, E3 +162640.472}
SPL {X  -162.820, Y  +392.460, Z    +0.000, E1   -17.627, E3 +162640.453}
SPL {X  -162.820, Y  +397.383, Z    +0.000, E1   -27.100, E3 +162640.523}
SPL {X  -162.820, Y  +404.822, Z    +0.000, E1   -40.113, E3 +162640.175}
SPL {X  -162.820, Y  +416.103, Z    +0.000, E1   -54.033, E3 +162640.027}
SPL {X  -162.820, Y  +472.592, Z    +0.000, E1   -70.190, E3 +162655.629}
SPL {X  -162.820, Y  +605.049, Z    +0.000, E1   -68.347, E3 +162750.111}
SPL {X  -162.820, Y  +616.480, Z    +0.000, E1   -67.752, E3 +162764.804}
SPL {X  -162.820, Y  +631.154, Z    +0.000, E1   -67.735, E3 +162777.338}
SPL {X  -162.820, Y  +647.590, Z    +0.000, E1   -67.861, E3 +162790.374}
SPL {X  -162.820, Y  +663.021, Z    +0.000, E1   -67.764, E3 +162804.211}
SPL {X  -162.642, Y  +681.112, Z    +0.000, E1   -67.812, E3 +162819.362}
SPL {X  -161.154, Y  +696.734, Z    +0.000, E1   -67.591, E3 +162834.359}
SPL {X  -158.503, Y  +710.744, Z    +0.000, E1   -67.284, E3 +162848.891}
SPL {X  -155.060, Y  +723.165, Z    +0.000, E1   -66.797, E3 +162863.067}
SPL {X  -151.511, Y  +733.123, Z    +0.000, E1   -66.286, E3 +162875.220}
SPL {X  -147.735, Y  +741.944, Z    +0.000, E1   -65.827, E3 +162885.747}
SPL {X  -144.196, Y  +749.116, Z    +0.000, E1   -65.203, E3 +162895.747}
SPL {X  -139.960, Y  +756.696, Z    +0.000, E1   -64.606, E3 +162905.641}
SPL {X  -135.604, Y  +763.621, Z    +0.000, E1   -63.883, E3 +162915.243}
SPL {X  -131.007, Y  +770.183, Z    +0.000, E1   -63.497, E3 +162922.528}
SPL {X   -85.750, Y  +811.910, Z    +0.000, E1   -55.921, E3 +163026.481}
ENDSPLINE

SPLINE
SPL {X  -114.463, Y  +789.295, Z    +0.000, E1   -54.865, E3 +163195.748}
SPL {X  -149.148, Y  +738.810, Z    +0.000, E1   -41.467, E3 +163206.819}
SPL {X  -159.693, Y  +705.258, Z    +0.000, E1   -25.118, E3 +163209.459}
SPL {X  -162.196, Y  +687.741, Z    +0.000, E1   -13.310, E3 +163210.424}
SPL {X  -162.791, Y  +676.596, Z    +0.000, E1    -4.586, E3 +163210.708}
SPL {X  -162.820, Y  +671.548, Z    +0.000, E1    -0.068, E3 +163210.185}
SPL {X  -162.820, Y  +669.949, Z    +0.000, E1    +2.213, E3 +163209.873}
SPL {X  -162.820, Y  +664.754, Z    +0.000, E1   +11.697, E3 +163209.772}
SPL {X  -162.820, Y  +658.944, Z    +0.000, E1   +23.544, E3 +163209.940}
SPL {X  -162.820, Y  +653.429, Z    +0.000, E1   +34.521, E3 +163209.330}
SPL {X  -162.820, Y  +647.179, Z    +0.000, E1   +44.317, E3 +163209.547}
SPL {X  -162.820, Y  +632.228, Z    +0.000, E1   +60.508, E3 +163208.667}
SPL {X  -162.820, Y  +572.535, Z    +0.000, E1   +70.270, E3 +163230.712}
SPL {X  -162.820, Y  +446.522, Z    +0.000, E1   +69.253, E3 +163314.536}
SPL {X  -162.820, Y  +444.665, Z    +0.000, E1   +68.107, E3 +163326.086}
SPL {X  -162.820, Y  +425.935, Z    +0.000, E1   +68.194, E3 +163341.141}
SPL {X  -162.820, Y  +405.187, Z    +0.000, E1   +68.161, E3 +163358.730}
SPL {X  -162.820, Y  +387.680, Z    +0.000, E1   +67.977, E3 +163374.918}
ENDSPLINE

SPLINE
SPL {X  -162.820, Y  +397.358, Z    +0.000, E1   +65.083, E3 +163389.557}
ENDSPLINE

SPLINE
SPL {X  -162.719, Y  +374.774, Z    +0.000, E1   +65.968, E3 +163404.041}
SPL {X  -160.017, Y  +350.416, Z    +0.000, E1   +67.091, E3 +163416.947}
SPL {X  -156.713, Y  +336.324, Z    +0.000, E1   +67.030, E3 +163429.543}
SPL {X  -153.279, Y  +325.584, Z    +0.000, E1   +66.662, E3 +163441.308}
SPL {X  -149.546, Y  +316.107, Z    +0.000, E1   +66.216, E3 +163452.484}
SPL {X  -147.033, Y  +310.560, Z    +0.000, E1   +65.497, E3 +163461.698}
SPL {X  -144.094, Y  +304.689, Z    +0.000, E1   +65.338, E3 +163467.710}
SPL {X  -141.093, Y  +299.241, Z    +0.000, E1   +65.039, E3 +163474.023}
SPL {X  -138.425, Y  +294.774, Z    +0.000, E1   +64.416, E3 +163481.207}
SPL {X  -134.374, Y  +288.555, Z    +0.000, E1   +63.758, E3 +163489.849}
SPL {X  -128.896, Y  +281.020, Z    +0.000, E1   +64.005, E3 +163494.972}
SPL {X   -85.291, Y  +241.807, Z    +0.000, E1   +53.957, E3 +163640.380}
ENDSPLINE

SPLINE
SPL {X  -136.861, Y  +292.299, Z    +0.000, E1   +47.815, E3 +163768.001}
SPL {X  -156.420, Y  +335.300, Z    +0.000, E1   +31.885, E3 +163775.790}
SPL {X  -161.293, Y  +358.252, Z    +0.000, E1   +18.542, E3 +163777.507}
SPL {X  -162.487, Y  +370.094, Z    +0.000, E1   +10.144, E3 +163777.585}
SPL {X  -162.818, Y  +379.612, Z    +0.000, E1    +2.663, E3 +163777.561}
SPL {X  -162.820, Y  +382.500, Z    +0.000, E1    +0.000, E3 +163777.154}
SPL {X  -162.820, Y  +383.629, Z    +0.000, E1    -1.565, E3 +163776.848}
SPL {X  -162.820, Y  +387.649, Z    +0.000, E1    -8.215, E3 +163776.836}
SPL {X  -162.820, Y  +392.460, Z    +0.000, E1   -17.627, E3 +163776.817}
SPL {X  -162.820, Y  +397.383, Z    +0.000, E1   -27.100, E3 +163776.887}
SPL {X  -162.820, Y  +404.822, Z    +0.000, E1   -40.113, E3 +163776.539}
SPL {X  -162.820, Y  +416.103, Z    +0.000, E1   -54.033, E3 +163776.391}
SPL {X  -162.820, Y  +472.592, Z    +0.000, E1   -70.190, E3 +163791.993}
SPL {X  -162.820, Y  +605.049, Z    +0.000, E1   -68.347, E3 +163886.474}
SPL {X  -162.820, Y  +616.480, Z    +0.000, E1   -67.752, E3 +163901.167}
SPL {X  -162.820, Y  +631.154, Z    +0.000, E1   -67.735, E3 +163913.702}
SPL {X  -162.820, Y  +647.590, Z    +0.000, E1   -67.861, E3 +163926.737}
SPL {X  -162.820, Y  +663.021, Z    +0.000, E1   -67.764, E3 +163940.575}
SPL {X  -162.799, Y  +676.123, Z    +0.000, E1   -67.801, E3 +163951.378}
SPL {X  -162.071, Y  +689.103, Z    +0.000, E1   -67.763, E3 +163962.785}
SPL {X  -160.908, Y  +698.381, Z    +0.000, E1   -67.466, E3 +163973.025}
SPL {X  -158.503, Y  +710.744, Z    +0.000, E1   -67.284, E3 +163985.254}
SPL {X  -155.060, Y  +723.165, Z    +0.000, E1   -66.797, E3 +163999.430}
SPL {X  -151.511, Y  +733.123, Z    +0.000, E1   -66.286, E3 +164011.584}
SPL {X  -148.440, Y  +740.403, Z    +0.000, E1   -65.944, E3 +164019.945}
SPL {X  -146.076, Y  +745.418, Z    +0.000, E1   -65.453, E3 +164027.420}
SPL {X  -142.207, Y  +752.793, Z    +0.000, E1   -65.028, E3 +164036.269}
SPL {X  -139.223, Y  +757.923, Z    +0.000, E1   -64.359, E3 +164044.239}
SPL {X  -135.604, Y  +763.621, Z    +0.000, E1   -63.883, E3 +164051.607}
SPL {X  -132.333, Y  +768.359, Z    +0.000, E1   -63.443, E3 +164057.575}
SPL {X  -129.515, Y  +772.172, Z    +0.000, E1   -63.535, E3 +164060.366}
SPL {X   -89.167, Y  +809.734, Z    +0.000, E1   -56.935, E3 +164145.784}
SPL {X   -81.104, Y  +814.683, Z    +0.000, E1   -54.328, E3 +164202.932}
ENDSPLINE

SPLINE
SPL {X  -114.463, Y  +789.295, Z    +0.000, E1   -54.865, E3 +164332.111}
SPL {X  -149.148, Y  +738.810, Z    +0.000, E1   -41.467, E3 +164343.183}
SPL {X  -159.693, Y  +705.258, Z    +0.000, E1   -25.118, E3 +164345.822}
SPL {X  -162.196, Y  +687.741, Z    +0.000, E1   -13.310, E3 +164346.787}
SPL {X  -162.791, Y  +676.596, Z    +0.000, E1    -4.586, E3 +164347.072}
SPL {X  -162.820, Y  +671.548, Z    +0.000, E1    -0.068, E3 +164346.549}
SPL {X  -162.820, Y  +669.949, Z    +0.000, E1    +2.213, E3 +164346.236}
SPL {X  -162.820, Y  +664.754, Z    +0.000, E1   +11.697, E3 +164346.135}
SPL {X  -162.820, Y  +658.944, Z    +0.000, E1   +23.544, E3 +164346.303}
SPL {X  -162.820, Y  +653.429, Z    +0.000, E1   +34.521, E3 +164345.694}
SPL {X  -162.820, Y  +647.179, Z    +0.000, E1   +44.317, E3 +164345.910}
SPL {X  -162.820, Y  +632.228, Z    +0.000, E1   +60.508, E3 +164345.031}
SPL {X  -162.820, Y  +572.535, Z    +0.000, E1   +70.270, E3 +164367.075}
SPL {X  -162.820, Y  +446.522, Z    +0.000, E1   +69.253, E3 +164450.899}
SPL {X  -162.820, Y  +444.665, Z    +0.000, E1   +68.107, E3 +164462.449}
SPL {X  -162.820, Y  +425.935, Z    +0.000, E1   +68.194, E3 +164477.505}
SPL {X  -162.820, Y  +409.792, Z    +0.000, E1   +68.121, E3 +164491.429}
SPL {X  -162.820, Y  +394.392, Z    +0.000, E1   +68.165, E3 +164504.003}
SPL {X  -162.820, Y  +385.264, Z    +0.000, E1   +67.766, E3 +164514.918}
ENDSPLINE

SPLINE
SPL {X  -162.820, Y  +401.104, Z    +0.000, E1   +65.023, E3 +164522.644}
ENDSPLINE

SPLINE
SPL {X  -162.820, Y  +386.513, Z    +0.000, E1   +65.423, E3 +164533.639}
SPL {X  -162.431, Y  +369.249, Z    +0.000, E1   +66.195, E3 +164543.641}
SPL {X  -160.017, Y  +350.416, Z    +0.000, E1   +67.091, E3 +164553.310}
SPL {X  -157.549, Y  +339.407, Z    +0.000, E1   +67.028, E3 +164563.187}
SPL {X  -154.848, Y  +330.175, Z    +0.000, E1   +66.891, E3 +164572.080}
SPL {X  -151.242, Y  +320.199, Z    +0.000, E1   +66.443, E3 +164583.881}
SPL {X  -147.540, Y  +311.636, Z    +0.000, E1   +65.718, E3 +164595.859}
SPL {X  -144.094, Y  +304.689, Z    +0.000, E1   +65.338, E3 +164604.074}
SPL {X  -141.093, Y  +299.241, Z    +0.000, E1   +65.039, E3 +164610.386}
SPL {X  -138.425, Y  +294.774, Z    +0.000, E1   +64.416, E3 +164617.570}
SPL {X  -135.581, Y  +290.344, Z    +0.000, E1   +63.996, E3 +164623.403}
SPL {X  -133.378, Y  +287.116, Z    +0.000, E1   +63.482, E3 +164628.567}
SPL {X  -128.896, Y  +281.020, Z    +0.000, E1   +64.005, E3 +164631.335}
SPL {X   -85.291, Y  +241.807, Z    +0.000, E1   +53.957, E3 +164776.743}
ENDSPLINE

SPLINE
SPL {X  -136.861, Y  +292.299, Z    +0.000, E1   +47.815, E3 +164904.364}
SPL {X  -156.420, Y  +335.300, Z    +0.000, E1   +31.885, E3 +164912.153}
SPL {X  -161.293, Y  +358.252, Z    +0.000, E1   +18.542, E3 +164913.871}
SPL {X  -162.687, Y  +373.932, Z    +0.000, E1    +7.306, E3 +164914.007}
SPL {X  -162.820, Y  +382.323, Z    +0.000, E1    +0.244, E3 +164913.566}
SPL {X  -162.820, Y  +383.629, Z    +0.000, E1    -1.565, E3 +164913.211}
SPL {X  -162.820, Y  +386.448, Z    +0.000, E1    -6.246, E3 +164913.157}
SPL {X  -162.820, Y  +391.031, Z    +0.000, E1   -14.627, E3 +164913.215}
SPL {X  -162.820, Y  +397.383, Z    +0.000, E1   -27.100, E3 +164913.251}
SPL {X  -162.820, Y  +404.822, Z    +0.000, E1   -40.113, E3 +164912.902}
SPL {X  -162.820, Y  +416.103, Z    +0.000, E1   -54.033, E3 +164912.754}
SPL {X  -162.820, Y  +472.592, Z    +0.000, E1   -70.190, E3 +164928.356}
SPL {X  -162.820, Y  +605.049, Z    +0.000, E1   -68.347, E3 +165022.838}
SPL {X  -162.820, Y  +616.480, Z    +0.000, E1   -67.752, E3 +165037.531}
SPL {X  -162.820, Y  +636.914, Z    +0.000, E1   -67.842, E3 +165054.225}
SPL {X  -162.820, Y  +654.663, Z    +0.000, E1   -67.744, E3 +165070.051}
SPL {X  -162.820, Y  +673.210, Z    +0.000, E1   -67.837, E3 +165085.084}
SPL {X  -162.071, Y  +689.103, Z    +0.000, E1   -67.763, E3 +165099.149}
SPL {X  -160.373, Y  +701.624, Z    +0.000, E1   -67.439, E3 +165112.508}
SPL {X  -157.887, Y  +713.277, Z    +0.000, E1   -67.197, E3 +165124.279}
SPL {X  -155.060, Y  +723.165, Z    +0.000, E1   -66.797, E3 +165135.794}
SPL {X  -152.159, Y  +731.448, Z    +0.000, E1   -66.356, E3 +165145.925}
SPL {X  -149.129, Y  +738.853, Z    +0.000, E1   -66.010, E3 +165154.622}
SPL {X  -146.076, Y  +745.418, Z    +0.000, E1   -65.453, E3 +165163.784}
SPL {X  -142.207, Y  +752.793, Z    +0.000, E1   -65.028, E3 +165172.632}
SPL {X  -139.223, Y  +757.923, Z    +0.000, E1   -64.359, E3 +165180.602}
SPL {X  -135.604, Y  +763.621, Z    +0.000, E1   -63.883, E3 +165187.970}
SPL {X  -131.007, Y  +770.183, Z    +0.000, E1   -63.497, E3 +165195.256}
SPL {X   -85.750, Y  +811.910, Z    +0.000, E1   -55.921, E3 +165299.208}
ENDSPLINE

SPLINE
SPL {X  -114.463, Y  +789.295, Z    +0.000, E1   -54.865, E3 +165468.475}
SPL {X  -149.148, Y  +738.810, Z    +0.000, E1   -41.467, E3 +165479.546}
SPL {X  -159.693, Y  +705.258, Z    +0.000, E1   -25.118, E3 +165482.186}
SPL {X  -162.196, Y  +687.741, Z    +0.000, E1   -13.310, E3 +165483.151}
SPL {X  -162.791, Y  +676.596, Z    +0.000, E1    -4.586, E3 +165483.435}
SPL {X  -162.820, Y  +671.385, Z    +0.000, E1    +0.078, E3 +165482.852}
SPL {X  -162.820, Y  +667.797, Z    +0.000, E1    +5.943, E3 +165482.511}
SPL {X  -162.820, Y  +663.306, Z    +0.000, E1   +14.820, E3 +165482.478}
SPL {X  -162.820, Y  +658.944, Z    +0.000, E1   +23.544, E3 +165482.667}
SPL {X  -162.820, Y  +650.349, Z    +0.000, E1   +39.427, E3 +165482.164}
SPL {X  -162.820, Y  +632.228, Z    +0.000, E1   +60.508, E3 +165481.394}
SPL {X  -162.820, Y  +572.535, Z    +0.000, E1   +70.270, E3 +165503.439}
SPL {X  -162.820, Y  +446.522, Z    +0.000, E1   +69.253, E3 +165587.263}
SPL {X  -162.820, Y  +444.665, Z    +0.000, E1   +68.107, E3 +165598.813}
SPL {X  -162.820, Y  +425.935, Z    +0.000, E1   +68.194, E3 +165613.869}
SPL {X  -162.820, Y  +409.792, Z    +0.000, E1   +68.121, E3 +165627.792}
SPL {X  -162.820, Y  +394.392, Z    +0.000, E1   +68.165, E3 +165640.367}
SPL {X  -162.820, Y  +385.264, Z    +0.000, E1   +67.766, E3 +165651.282}
ENDSPLINE

SPLINE
SPL {X  -162.820, Y  +401.104, Z    +0.000, E1   +65.023, E3 +165659.008}
ENDSPLINE

SPLINE
SPL {X  -162.820, Y  +386.513, Z    +0.000, E1   +65.423, E3 +165670.003}
SPL {X  -162.431, Y  +369.249, Z    +0.000, E1   +66.195, E3 +165680.004}
SPL {X  -160.017, Y  +350.416, Z    +0.000, E1   +67.091, E3 +165689.674}
SPL {X  -157.549, Y  +339.407, Z    +0.000, E1   +67.028, E3 +165699.550}
SPL {X  -154.848, Y  +330.175, Z    +0.000, E1   +66.891, E3 +165708.443}
SPL {X  -151.242, Y  +320.199, Z    +0.000, E1   +66.443, E3 +165720.244}
SPL {X  -147.540, Y  +311.636, Z    +0.000, E1   +65.718, E3 +165732.223}
SPL {X  -144.094, Y  +304.689, Z    +0.000, E1   +65.338, E3 +165740.437}
SPL {X  -141.093, Y  +299.241, Z    +0.000, E1   +65.039, E3 +165746.750}
SPL {X  -138.425, Y  +294.774, Z    +0.000, E1   +64.416, E3 +165753.934}
SPL {X  -135.581, Y  +290.344, Z    +0.000, E1   +63.996, E3 +165759.766}
SPL {X  -133.378, Y  +287.116, Z    +0.000, E1   +63.482, E3 +165764.930}
SPL {X  -128.896, Y  +281.020, Z    +0.000, E1   +64.005, E3 +165767.699}
SPL {X   -85.291, Y  +241.807, Z    +0.000, E1   +53.957, E3 +165913.107}
ENDSPLINE

SPLINE
SPL {X  -136.861, Y  +292.299, Z    +0.000, E1   +47.815, E3 +166040.728}
SPL {X  -156.420, Y  +335.300, Z    +0.000, E1   +31.885, E3 +166048.517}
SPL {X  -161.293, Y  +358.252, Z    +0.000, E1   +18.542, E3 +166050.234}
SPL {X  -162.487, Y  +370.094, Z    +0.000, E1   +10.144, E3 +166050.313}
SPL {X  -162.818, Y  +379.612, Z    +0.000, E1    +2.663, E3 +166050.288}
SPL {X  -162.820, Y  +382.500, Z    +0.000, E1    +0.000, E3 +166049.882}
SPL {X  -162.820, Y  +383.629, Z    +0.000, E1    -1.565, E3 +166049.575}
SPL {X  -162.820, Y  +386.448, Z    +0.000, E1    -6.246, E3 +166049.520}
SPL {X  -162.820, Y  +391.031, Z    +0.000, E1   -14.627, E3 +166049.579}
SPL {X  -162.820, Y  +397.383, Z    +0.000, E1   -27.100, E3 +166049.614}
SPL {X  -162.820, Y  +404.822, Z    +0.000, E1   -40.113, E3 +166049.266}
SPL {X  -162.820, Y  +416.103, Z    +0.000, E1   -54.033, E3 +166049.118}
SPL {X  -162.820, Y  +467.510, Z    +0.000, E1   -69.867, E3 +166062.696}
SPL {X  -162.820, Y  +604.717, Z    +0.000, E1   -70.047, E3 +166144.416}
SPL {X  -162.820, Y  +606.663, Z    +0.000, E1   -67.762, E3 +166165.464}
SPL {X  -162.820, Y  +626.641, Z    +0.000, E1   -67.759, E3 +166182.571}
SPL {X  -162.820, Y  +643.417, Z    +0.000, E1   -67.904, E3 +166195.388}
SPL {X  -162.820, Y  +654.663, Z    +0.000, E1   -67.744, E3 +166206.414}
SPL {X  -162.820, Y  +673.210, Z    +0.000, E1   -67.837, E3 +166221.448}
SPL {X  -162.071, Y  +689.103, Z    +0.000, E1   -67.763, E3 +166235.513}
SPL {X  -160.908, Y  +698.381, Z    +0.000, E1   -67.466, E3 +166245.752}
SPL {X  -158.503, Y  +710.744, Z    +0.000, E1   -67.284, E3 +166257.981}
SPL {X  -155.060, Y  +723.165, Z    +0.000, E1   -66.797, E3 +166272.158}
SPL {X  -151.511, Y  +733.123, Z    +0.000, E1   -66.286, E3 +166284.311}
SPL {X  -148.440, Y  +740.403, Z    +0.000, E1   -65.944, E3 +166292.672}
SPL {X  -146.076, Y  +745.418, Z    +0.000, E1   -65.453, E3 +166300.147}
SPL {X  -142.207, Y  +752.793, Z    +0.000, E1   -65.028, E3 +166308.996}
SPL {X  -139.223, Y  +757.923, Z    +0.000, E1   -64.359, E3 +166316.966}
SPL {X  -135.604, Y  +763.621, Z    +0.000, E1   -63.883, E3 +166324.334}
SPL {X  -131.007, Y  +770.183, Z    +0.000, E1   -63.497, E3 +166331.619}
SPL {X   -85.750, Y  +811.910, Z    +0.000, E1   -55.921, E3 +166435.572}
ENDSPLINE

SPLINE
SPL {X  -114.463, Y  +789.295, Z    +0.000, E1   -54.865, E3 +166604.839}
SPL {X  -144.553, Y  +748.431, Z    +0.000, E1   -44.979, E3 +166615.547}
SPL {X  -156.024, Y  +720.050, Z    +0.000, E1   -33.178, E3 +166617.113}
SPL {X  -160.714, Y  +699.606, Z    +0.000, E1   -21.520, E3 +166618.987}
SPL {X  -162.196, Y  +687.741, Z    +0.000, E1   -13.310, E3 +166619.515}
SPL {X  -162.791, Y  +676.596, Z    +0.000, E1    -4.586, E3 +166619.799}
SPL {X  -162.820, Y  +671.548, Z    +0.000, E1    -0.068, E3 +166619.276}
SPL {X  -162.820, Y  +669.949, Z    +0.000, E1    +2.213, E3 +166618.964}
SPL {X  -162.820, Y  +664.754, Z    +0.000, E1   +11.697, E3 +166618.863}
SPL {X  -162.820, Y  +658.944, Z    +0.000, E1   +23.544, E3 +166619.031}
SPL {X  -162.820, Y  +650.349, Z    +0.000, E1   +39.427, E3 +166618.528}
SPL {X  -162.820, Y  +632.228, Z    +0.000, E1   +60.508, E3 +166617.758}
SPL {X  -162.820, Y  +572.535, Z    +0.000, E1   +70.270, E3 +166639.803}
SPL {X  -162.820, Y  +446.522, Z    +0.000, E1   +69.253, E3 +166723.626}
SPL {X  -162.820, Y  +440.686, Z    +0.000, E1   +68.127, E3 +166738.501}
SPL {X  -162.820, Y  +421.575, Z    +0.000, E1   +68.212, E3 +166753.565}
SPL {X  -162.820, Y  +409.792, Z    +0.000, E1   +68.121, E3 +166764.156}
SPL {X  -162.820, Y  +394.392, Z    +0.000, E1   +68.165, E3 +166776.730}
SPL {X  -162.820, Y  +385.264, Z    +0.000, E1   +67.766, E3 +166787.646}
ENDSPLINE

SPLINE
SPL {X  -162.820, Y  +401.104, Z    +0.000, E1   +65.023, E3 +166795.371}
ENDSPLINE

SPLINE
SPL {X  -162.820, Y  +386.513, Z    +0.000, E1   +65.423, E3 +166806.367}
SPL {X  -162.431, Y  +369.249, Z    +0.000, E1   +66.195, E3 +166816.368}
SPL {X  -160.017, Y  +350.416, Z    +0.000, E1   +67.091, E3 +166826.038}
SPL {X  -156.713, Y  +336.324, Z    +0.000, E1   +67.030, E3 +166838.634}
SPL {X  -153.279, Y  +325.584, Z    +0.000, E1   +66.662, E3 +166850.399}
SPL {X  -149.546, Y  +316.107, Z    +0.000, E1   +66.216, E3 +166861.575}
SPL {X  -147.033, Y  +310.560, Z    +0.000, E1   +65.497, E3 +166870.789}
SPL {X  -144.094, Y  +304.689, Z    +0.000, E1   +65.338, E3 +166876.801}
SPL {X  -141.093, Y  +299.241, Z    +0.000, E1   +65.039, E3 +166883.114}
SPL {X  -138.425, Y  +294.774, Z    +0.000, E1   +64.416, E3 +166890.297}
SPL {X  -134.374, Y  +288.555, Z    +0.000, E1   +63.758, E3 +166898.940}
SPL {X  -128.896, Y  +281.020, Z    +0.000, E1   +64.005, E3 +166904.063}
SPL {X   -85.291, Y  +241.807, Z    +0.000, E1   +53.957, E3 +167049.471}
ENDSPLINE

SPLINE
SPL {X  -136.861, Y  +292.299, Z    +0.000, E1   +47.815, E3 +167177.091}
SPL {X  -156.420, Y  +335.300, Z    +0.000, E1   +31.885, E3 +167184.881}
SPL {X  -161.293, Y  +358.252, Z    +0.000, E1   +18.542, E3 +167186.598}
SPL {X  -162.487, Y  +370.094, Z    +0.000, E1   +10.144, E3 +167186.676}
SPL {X  -162.818, Y  +379.612, Z    +0.000, E1    +2.663, E3 +167186.652}
SPL {X  -162.820, Y  +382.500, Z    +0.000, E1    +0.000, E3 +167186.245}
SPL {X  -162.820, Y  +383.629, Z    +0.000, E1    -1.565, E3 +167185.939}
SPL {X  -162.820, Y  +387.649, Z    +0.000, E1    -8.215, E3 +167185.926}
SPL {X  -162.820, Y  +392.460, Z    +0.000, E1   -17.627, E3 +167185.908}
SPL {X  -162.820, Y  +397.383, Z    +0.000, E1   -27.100, E3 +167185.978}
SPL {X  -162.820, Y  +404.822, Z    +0.000, E1   -40.113, E3 +167185.630}
SPL {X  -162.820, Y  +416.103, Z    +0.000, E1   -54.033, E3 +167185.482}
SPL {X  -162.820, Y  +467.510, Z    +0.000, E1   -69.867, E3 +167199.060}
SPL {X  -162.820, Y  +604.717, Z    +0.000, E1   -70.047, E3 +167280.779}
SPL {X  -162.820, Y  +606.663, Z    +0.000, E1   -67.762, E3 +167301.828}
SPL {X  -162.820, Y  +626.641, Z    +0.000, E1   -67.759, E3 +167318.935}
SPL {X  -162.820, Y  +647.590, Z    +0.000, E1   -67.861, E3 +167335.828}
SPL {X  -162.820, Y  +663.021, Z    +0.000, E1   -67.764, E3 +167349.666}
SPL {X  -162.799, Y  +676.123, Z    +0.000, E1   -67.801, E3 +167360.469}
SPL {X  -162.071, Y  +689.103, Z    +0.000, E1   -67.763, E3 +167371.876}
SPL {X  -160.373, Y  +701.624, Z    +0.000, E1   -67.439, E3 +167385.235}
SPL {X  -157.320, Y  +715.461, Z    +0.000, E1   -67.133, E3 +167399.514}
SPL {X  -154.452, Y  +725.025, Z    +0.000, E1   -66.701, E3 +167410.699}
SPL {X  -152.159, Y  +731.448, Z    +0.000, E1   -66.356, E3 +167418.652}
SPL {X  -148.374, Y  +740.549, Z    +0.000, E1   -65.919, E3 +167429.526}
SPL {X  -144.196, Y  +749.116, Z    +0.000, E1   -65.203, E3 +167441.201}
SPL {X  -141.115, Y  +754.722, Z    +0.000, E1   -64.893, E3 +167447.661}
SPL {X  -138.151, Y  +759.667, Z    +0.000, E1   -64.251, E3 +167455.483}
SPL {X  -134.751, Y  +764.892, Z    +0.000, E1   -63.716, E3 +167462.485}
SPL {X  -131.007, Y  +770.183, Z    +0.000, E1   -63.497, E3 +167467.983}
SPL {X   -85.750, Y  +811.910, Z    +0.000, E1   -55.921, E3 +167571.935}
ENDSPLINE

SPLINE
SPL {X  -114.463, Y  +789.295, Z    +0.000, E1   -54.865, E3 +167741.202}
SPL {X  -144.553, Y  +748.431, Z    +0.000, E1   -44.979, E3 +167751.911}
SPL {X  -156.024, Y  +720.050, Z    +0.000, E1   -33.178, E3 +167753.477}
SPL {X  -160.714, Y  +699.606, Z    +0.000, E1   -21.520, E3 +167755.351}
SPL {X  -162.196, Y  +687.741, Z    +0.000, E1   -13.310, E3 +167755.878}
SPL {X  -162.791, Y  +676.596, Z    +0.000, E1    -4.586, E3 +167756.163}
SPL {X  -162.820, Y  +671.548, Z    +0.000, E1    -0.068, E3 +167755.640}
SPL {X  -162.820, Y  +669.949, Z    +0.000, E1    +2.213, E3 +167755.327}
SPL {X  -162.820, Y  +664.754, Z    +0.000, E1   +11.697, E3 +167755.226}
SPL {X  -162.820, Y  +658.944, Z    +0.000, E1   +23.544, E3 +167755.394}
SPL {X  -162.820, Y  +650.349, Z    +0.000, E1   +39.427, E3 +167754.891}
SPL {X  -162.820, Y  +635.494, Z    +0.000, E1   +57.613, E3 +167754.594}
SPL {X  -162.820, Y  +626.637, Z    +0.000, E1   +64.941, E3 +167753.310}
SPL {X  -162.820, Y  +572.535, Z    +0.000, E1   +70.270, E3 +167776.166}
SPL {X  -162.820, Y  +446.522, Z    +0.000, E1   +69.253, E3 +167859.990}
SPL {X  -162.820, Y  +444.665, Z    +0.000, E1   +68.107, E3 +167871.540}
SPL {X  -162.820, Y  +425.935, Z    +0.000, E1   +68.194, E3 +167886.596}
SPL {X  -162.820, Y  +405.187, Z    +0.000, E1   +68.161, E3 +167904.184}
SPL {X  -162.820, Y  +387.680, Z    +0.000, E1   +67.977, E3 +167920.373}
ENDSPLINE

SPLINE
SPL {X  -162.820, Y  +397.358, Z    +0.000, E1   +65.083, E3 +167935.011}
ENDSPLINE

SPLINE
SPL {X  -162.719, Y  +374.774, Z    +0.000, E1   +65.968, E3 +167949.496}
SPL {X  -160.017, Y  +350.416, Z    +0.000, E1   +67.091, E3 +167962.401}
SPL {X  -157.549, Y  +339.407, Z    +0.000, E1   +67.028, E3 +167972.277}
SPL {X  -154.848, Y  +330.175, Z    +0.000, E1   +66.891, E3 +167981.170}
SPL {X  -151.242, Y  +320.199, Z    +0.000, E1   +66.443, E3 +167992.972}
SPL {X  -147.540, Y  +311.636, Z    +0.000, E1   +65.718, E3 +168004.950}
SPL {X  -144.094, Y  +304.689, Z    +0.000, E1   +65.338, E3 +168013.164}
SPL {X  -141.093, Y  +299.241, Z    +0.000, E1   +65.039, E3 +168019.477}
SPL {X  -138.425, Y  +294.774, Z    +0.000, E1   +64.416, E3 +168026.661}
SPL {X  -134.374, Y  +288.555, Z    +0.000, E1   +63.758, E3 +168035.303}
SPL {X  -128.896, Y  +281.020, Z    +0.000, E1   +64.005, E3 +168040.426}
SPL {X   -85.291, Y  +241.807, Z    +0.000, E1   +53.957, E3 +168185.834}
ENDSPLINE

SPLINE
SPL {X  -136.861, Y  +292.299, Z    +0.000, E1   +47.815, E3 +168313.455}
SPL {X  -152.886, Y  +324.498, Z    +0.000, E1   +36.840, E3 +168320.137}
SPL {X  -158.256, Y  +342.219, Z    +0.000, E1   +28.198, E3 +168321.770}
SPL {X  -161.293, Y  +358.252, Z    +0.000, E1   +18.542, E3 +168322.962}
SPL {X  -162.687, Y  +373.932, Z    +0.000, E1    +7.306, E3 +168323.097}
SPL {X  -162.820, Y  +382.323, Z    +0.000, E1    +0.244, E3 +168322.656}
SPL {X  -162.820, Y  +383.629, Z    +0.000, E1    -1.565, E3 +168322.302}
SPL {X  -162.820, Y  +386.448, Z    +0.000, E1    -6.246, E3 +168322.248}
SPL {X  -162.820, Y  +391.031, Z    +0.000, E1   -14.627, E3 +168322.306}
SPL {X  -162.820, Y  +397.383, Z    +0.000, E1   -27.100, E3 +168322.342}
SPL {X  -162.820, Y  +404.822, Z    +0.000, E1   -40.113, E3 +168321.993}
SPL {X  -162.820, Y  +416.103, Z    +0.000, E1   -54.033, E3 +168321.845}
SPL {X  -162.820, Y  +467.510, Z    +0.000, E1   -69.867, E3 +168335.423}
SPL {X  -162.820, Y  +604.717, Z    +0.000, E1   -70.047, E3 +168417.143}
ENDSPLINE

SPLINE
SPL {X  -162.820, Y  +602.324, Z    +0.000, E1   -67.733, E3 +168434.592}
ENDSPLINE

SPLINE
SPL {X  -162.820, Y  +616.480, Z    +0.000, E1   -67.752, E3 +168446.622}
SPL {X  -162.820, Y  +636.914, Z    +0.000, E1   -67.842, E3 +168463.316}
SPL {X  -162.820, Y  +651.339, Z    +0.000, E1   -67.768, E3 +168475.984}
SPL {X  -162.820, Y  +663.021, Z    +0.000, E1   -67.764, E3 +168486.029}
SPL {X  -162.642, Y  +681.112, Z    +0.000, E1   -67.812, E3 +168501.181}
SPL {X  -161.154, Y  +696.734, Z    +0.000, E1   -67.591, E3 +168516.178}
SPL {X  -158.503, Y  +710.744, Z    +0.000, E1   -67.284, E3 +168530.709}
SPL {X  -155.060, Y  +723.165, Z    +0.000, E1   -66.797, E3 +168544.885}
SPL {X  -152.159, Y  +731.448, Z    +0.000, E1   -66.356, E3 +168555.016}
SPL {X  -149.129, Y  +738.853, Z    +0.000, E1   -66.010, E3 +168563.713}
SPL {X  -146.076, Y  +745.418, Z    +0.000, E1   -65.453, E3 +168572.874}
SPL {X  -143.238, Y  +750.916, Z    +0.000, E1   -65.112, E3 +168579.559}
SPL {X  -139.960, Y  +756.696, Z    +0.000, E1   -64.606, E3 +168587.459}
SPL {X  -135.604, Y  +763.621, Z    +0.000, E1   -63.883, E3 +168597.061}
SPL {X  -132.333, Y  +768.359, Z    +0.000, E1   -63.443, E3 +168603.030}
SPL {X  -129.515, Y  +772.172, Z    +0.000, E1   -63.535, E3 +168605.821}
SPL {X   -85.750, Y  +811.910, Z    +0.000, E1   -55.921, E3 +168708.299}
ENDSPLINE

SPLINE
SPL {X  -114.463, Y  +789.295, Z    +0.000, E1   -54.865, E3 +168877.566}
SPL {X  -144.553, Y  +748.431, Z    +0.000, E1   -44.979, E3 +168888.274}
SPL {X  -156.024, Y  +720.050, Z    +0.000, E1   -33.178, E3 +168889.841}
SPL {X  -160.714, Y  +699.606, Z    +0.000, E1   -21.520, E3 +168891.715}
SPL {X  -162.196, Y  +687.741, Z    +0.000, E1   -13.310, E3 +168892.242}
SPL {X  -162.791, Y  +676.596, Z    +0.000, E1    -4.586, E3 +168892.526}
SPL {X  -162.820, Y  +671.548, Z    +0.000, E1    -0.068, E3 +168892.003}
SPL {X  -162.820, Y  +669.949, Z    +0.000, E1    +2.213, E3 +168891.691}
SPL {X  -162.820, Y  +664.754, Z    +0.000, E1   +11.697, E3 +168891.590}
SPL {X  -162.820, Y  +658.944, Z    +0.000, E1   +23.544, E3 +168891.758}
SPL {X  -162.820, Y  +650.349, Z    +0.000, E1   +39.427, E3 +168891.255}
SPL {X  -162.820, Y  +632.228, Z    +0.000, E1   +60.508, E3 +168890.485}
SPL {X  -162.820, Y  +572.535, Z    +0.000, E1   +70.270, E3 +168912.530}
SPL {X  -162.820, Y  +446.522, Z    +0.000, E1   +69.253, E3 +168996.354}
SPL {X  -162.820, Y  +440.686, Z    +0.000, E1   +68.127, E3 +169011.228}
SPL {X  -162.820, Y  +421.575, Z    +0.000, E1   +68.212, E3 +169026.292}
SPL {X  -162.820, Y  +409.792, Z    +0.000, E1   +68.121, E3 +169036.883}
SPL {X  -162.820, Y  +394.392, Z    +0.000, E1   +68.165, E3 +169049.458}
SPL {X  -162.820, Y  +385.264, Z    +0.000, E1   +67.766, E3 +169060.373}
ENDSPLINE

SPLINE
SPL {X  -162.820, Y  +401.104, Z    +0.000, E1   +65.023, E3 +169068.098}
ENDSPLINE

SPLINE
SPL {X  -162.820, Y  +386.513, Z    +0.000, E1   +65.423, E3 +169079.094}
SPL {X  -162.431, Y  +369.249, Z    +0.000, E1   +66.195, E3 +169089.095}
SPL {X  -160.017, Y  +350.416, Z    +0.000, E1   +67.091, E3 +169098.765}
SPL {X  -156.713, Y  +336.324, Z    +0.000, E1   +67.030, E3 +169111.361}
SPL {X  -153.279, Y  +325.584, Z    +0.000, E1   +66.662, E3 +169123.126}
SPL {X  -149.546, Y  +316.107, Z    +0.000, E1   +66.216, E3 +169134.302}
SPL {X  -147.033, Y  +310.560, Z    +0.000, E1   +65.497, E3 +169143.516}
SPL {X  -144.094, Y  +304.689, Z    +0.000, E1   +65.338, E3 +169149.528}
SPL {X  -141.093, Y  +299.241, Z    +0.000, E1   +65.039, E3 +169155.841}
SPL {X  -138.425, Y  +294.774, Z    +0.000, E1   +64.416, E3 +169163.025}
SPL {X  -135.581, Y  +290.344, Z    +0.000, E1   +63.996, E3 +169168.857}
SPL {X  -132.317, Y  +285.618, Z    +0.000, E1   +63.461, E3 +169175.432}
SPL {X  -126.028, Y  +277.411, Z    +0.000, E1   +65.004, E3 +169175.604}
SPL {X   -85.291, Y  +241.807, Z    +0.000, E1   +53.957, E3 +169322.198}
ENDSPLINE

SPLINE
SPL {X  -136.861, Y  +292.299, Z    +0.000, E1   +47.815, E3 +169449.819}
SPL {X  -156.420, Y  +335.300, Z    +0.000, E1   +31.885, E3 +169457.608}
SPL {X  -161.293, Y  +358.252, Z    +0.000, E1   +18.542, E3 +169459.325}
SPL {X  -162.487, Y  +370.094, Z    +0.000, E1   +10.144, E3 +169459.404}
SPL {X  -162.818, Y  +379.612, Z    +0.000, E1    +2.663, E3 +169459.379}
SPL {X  -162.820, Y  +382.500, Z    +0.000, E1    +0.000, E3 +169458.973}
SPL {X  -162.820, Y  +383.629, Z    +0.000, E1    -1.565, E3 +169458.666}
SPL {X  -162.820, Y  +387.649, Z    +0.000, E1    -8.215, E3 +169458.654}
SPL {X  -162.820, Y  +392.460, Z    +0.000, E1   -17.627, E3 +169458.635}
SPL {X  -162.820, Y  +397.383, Z    +0.000, E1   -27.100, E3 +169458.705}
SPL {X  -162.820, Y  +404.822, Z    +0.000, E1   -40.113, E3 +169458.357}
SPL {X  -162.820, Y  +416.103, Z    +0.000, E1   -54.033, E3 +169458.209}
SPL {X  -162.820, Y  +472.592, Z    +0.000, E1   -70.190, E3 +169473.811}
SPL {X  -162.820, Y  +605.049, Z    +0.000, E1   -68.347, E3 +169568.293}
SPL {X  -162.820, Y  +616.480, Z    +0.000, E1   -67.752, E3 +169582.986}
SPL {X  -162.820, Y  +631.154, Z    +0.000, E1   -67.735, E3 +169595.520}
SPL {X  -162.820, Y  +647.590, Z    +0.000, E1   -67.861, E3 +169608.555}
SPL {X  -162.820, Y  +663.021, Z    +0.000, E1   -67.764, E3 +169622.393}
SPL {X  -162.642, Y  +681.112, Z    +0.000, E1   -67.812, E3 +169637.544}
SPL {X  -161.154, Y  +696.734, Z    +0.000, E1   -67.591, E3 +169652.541}
SPL {X  -158.503, Y  +710.744, Z    +0.000, E1   -67.284, E3 +169667.072}
SPL {X  -155.060, Y  +723.165, Z    +0.000, E1   -66.797, E3 +169681.248}
SPL {X  -151.511, Y  +733.123, Z    +0.000, E1   -66.286, E3 +169693.402}
SPL {X  -147.735, Y  +741.944, Z    +0.000, E1   -65.827, E3 +169703.928}
SPL {X  -144.196, Y  +749.116, Z    +0.000, E1   -65.203, E3 +169713.929}
SPL {X  -139.960, Y  +756.696, Z    +0.000, E1   -64.606, E3 +169723.823}
SPL {X  -135.604, Y  +763.621, Z    +0.000, E1   -63.883, E3 +169733.425}
SPL {X  -131.007, Y  +770.183, Z    +0.000, E1   -63.497, E3 +169740.710}
SPL {X   -85.750, Y  +811.910, Z    +0.000, E1   -55.921, E3 +169844.663}
ENDSPLINE

SPLINE
SPL {X  -114.463, Y  +789.295, Z    +0.000, E1   -54.865, E3 +170013.930}
SPL {X  -149.148, Y  +738.810, Z    +0.000, E1   -41.467, E3 +170025.001}
SPL {X  -159.693, Y  +705.258, Z    +0.000, E1   -25.118, E3 +170027.640}
SPL {X  -162.196, Y  +687.741, Z    +0.000, E1   -13.310, E3 +170028.606}
SPL {X  -162.791, Y  +676.596, Z    +0.000, E1    -4.586, E3 +170028.890}
SPL {X  -162.820, Y  +671.548, Z    +0.000, E1    -0.068, E3 +170028.367}
SPL {X  -162.820, Y  +669.949, Z    +0.000, E1    +2.213, E3 +170028.054}
SPL {X  -162.820, Y  +664.754, Z    +0.000, E1   +11.697, E3 +170027.953}
SPL {X  -162.820, Y  +658.944, Z    +0.000, E1   +23.544, E3 +170028.122}
SPL {X  -162.820, Y  +653.429, Z    +0.000, E1   +34.521, E3 +170027.512}
SPL {X  -162.820, Y  +647.179, Z    +0.000, E1   +44.317, E3 +170027.729}
SPL {X  -162.820, Y  +632.228, Z    +0.000, E1   +60.508, E3 +170026.849}
SPL {X  -162.820, Y  +572.535, Z    +0.000, E1   +70.270, E3 +170048.893}
SPL {X  -162.820, Y  +446.522, Z    +0.000, E1   +69.253, E3 +170132.717}
SPL {X  -162.820, Y  +440.686, Z    +0.000, E1   +68.127, E3 +170147.592}
SPL {X  -162.820, Y  +421.575, Z    +0.000, E1   +68.212, E3 +170162.656}
SPL {X  -162.820, Y  +409.792, Z    +0.000, E1   +68.121, E3 +170173.247}
SPL {X  -162.820, Y  +394.392, Z    +0.000, E1   +68.165, E3 +170185.821}
SPL {X  -162.820, Y  +385.264, Z    +0.000, E1   +67.766, E3 +170196.737}
ENDSPLINE

SPLINE
SPL {X  -162.820, Y  +401.104, Z    +0.000, E1   +65.023, E3 +170204.462}
ENDSPLINE

SPLINE
SPL {X  -162.820, Y  +386.513, Z    +0.000, E1   +65.423, E3 +170215.457}
SPL {X  -161.886, Y  +363.082, Z    +0.000, E1   +66.474, E3 +170228.890}
SPL {X  -158.043, Y  +341.350, Z    +0.000, E1   +67.216, E3 +170242.086}
SPL {X  -154.848, Y  +330.175, Z    +0.000, E1   +66.891, E3 +170253.898}
SPL {X  -152.657, Y  +323.878, Z    +0.000, E1   +66.551, E3 +170261.632}
SPL {X  -149.546, Y  +316.107, Z    +0.000, E1   +66.216, E3 +170270.666}
SPL {X  -147.033, Y  +310.560, Z    +0.000, E1   +65.497, E3 +170279.880}
SPL {X  -144.094, Y  +304.689, Z    +0.000, E1   +65.338, E3 +170285.892}
SPL {X  -141.093, Y  +299.241, Z    +0.000, E1   +65.039, E3 +170292.204}
SPL {X  -138.425, Y  +294.774, Z    +0.000, E1   +64.416, E3 +170299.388}
SPL {X  -134.374, Y  +288.555, Z    +0.000, E1   +63.758, E3 +170308.031}
SPL {X  -128.896, Y  +281.020, Z    +0.000, E1   +64.005, E3 +170313.153}
SPL {X   -85.291, Y  +241.807, Z    +0.000, E1   +53.957, E3 +170458.561}
ENDSPLINE

SPLINE
SPL {X  -136.861, Y  +292.299, Z    +0.000, E1   +47.815, E3 +170586.182}
SPL {X  -156.420, Y  +335.300, Z    +0.000, E1   +31.885, E3 +170593.972}
SPL {X  -161.293, Y  +358.252, Z    +0.000, E1   +18.542, E3 +170595.689}
SPL {X  -162.487, Y  +370.094, Z    +0.000, E1   +10.144, E3 +170595.767}
SPL {X  -162.818, Y  +379.612, Z    +0.000, E1    +2.663, E3 +170595.743}
SPL {X  -162.820, Y  +382.500, Z    +0.000, E1    +0.000, E3 +170595.336}
SPL {X  -162.820, Y  +383.629, Z    +0.000, E1    -1.565, E3 +170595.029}
SPL {X  -162.820, Y  +387.649, Z    +0.000, E1    -8.215, E3 +170595.017}
SPL {X  -162.820, Y  +392.460, Z    +0.000, E1   -17.627, E3 +170594.999}
SPL {X  -162.820, Y  +397.383, Z    +0.000, E1   -27.100, E3 +170595.069}
SPL {X  -162.820, Y  +404.822, Z    +0.000, E1   -40.113, E3 +170594.720}
SPL {X  -162.820, Y  +416.103, Z    +0.000, E1   -54.033, E3 +170594.573}
SPL {X  -162.820, Y  +467.510, Z    +0.000, E1   -69.867, E3 +170608.151}
SPL {X  -162.820, Y  +604.717, Z    +0.000, E1   -70.047, E3 +170689.870}
ENDSPLINE

SPLINE
SPL {X  -162.820, Y  +602.324, Z    +0.000, E1   -67.733, E3 +170707.319}
ENDSPLINE

SPLINE
SPL {X  -162.820, Y  +616.480, Z    +0.000, E1   -67.752, E3 +170719.349}
SPL {X  -162.820, Y  +636.914, Z    +0.000, E1   -67.842, E3 +170736.043}
SPL {X  -162.820, Y  +654.663, Z    +0.000, E1   -67.744, E3 +170751.869}
SPL {X  -162.820, Y  +673.210, Z    +0.000, E1   -67.837, E3 +170766.902}
SPL {X  -162.071, Y  +689.103, Z    +0.000, E1   -67.763, E3 +170780.967}
SPL {X  -160.373, Y  +701.624, Z    +0.000, E1   -67.439, E3 +170794.326}
SPL {X  -157.887, Y  +713.277, Z    +0.000, E1   -67.197, E3 +170806.098}
SPL {X  -155.060, Y  +723.165, Z    +0.000, E1   -66.797, E3 +170817.612}
SPL {X  -151.511, Y  +733.123, Z    +0.000, E1   -66.286, E3 +170829.766}
SPL {X  -147.735, Y  +741.944, Z    +0.000, E1   -65.827, E3 +170840.292}
SPL {X  -144.196, Y  +749.116, Z    +0.000, E1   -65.203, E3 +170850.292}
SPL {X  -139.960, Y  +756.696, Z    +0.000, E1   -64.606, E3 +170860.187}
SPL {X  -135.604, Y  +763.621, Z    +0.000, E1   -63.883, E3 +170869.789}
SPL {X  -131.007, Y  +770.183, Z    +0.000, E1   -63.497, E3 +170877.074}
SPL {X   -85.750, Y  +811.910, Z    +0.000, E1   -55.921, E3 +170981.026}
ENDSPLINE

SPLINE
SPL {X  -114.463, Y  +789.295, Z    +0.000, E1   -54.865, E3 +171150.293}
SPL {X  -149.148, Y  +738.810, Z    +0.000, E1   -41.467, E3 +171161.364}
SPL {X  -159.693, Y  +705.258, Z    +0.000, E1   -25.118, E3 +171164.004}
SPL {X  -162.196, Y  +687.741, Z    +0.000, E1   -13.310, E3 +171164.969}
SPL {X  -162.791, Y  +676.596, Z    +0.000, E1    -4.586, E3 +171165.253}
SPL {X  -162.820, Y  +671.385, Z    +0.000, E1    +0.078, E3 +171164.671}
SPL {X  -162.820, Y  +667.797, Z    +0.000, E1    +5.943, E3 +171164.329}
SPL {X  -162.820, Y  +663.306, Z    +0.000, E1   +14.820, E3 +171164.296}
SPL {X  -162.820, Y  +658.944, Z    +0.000, E1   +23.544, E3 +171164.485}
SPL {X  -162.820, Y  +650.349, Z    +0.000, E1   +39.427, E3 +171163.982}
SPL {X  -162.820, Y  +632.228, Z    +0.000, E1   +60.508, E3 +171163.212}
SPL {X  -162.820, Y  +572.535, Z    +0.000, E1   +70.270, E3 +171185.257}
SPL {X  -162.820, Y  +446.522, Z    +0.000, E1   +69.253, E3 +171269.081}
SPL {X  -162.820, Y  +444.665, Z    +0.000, E1   +68.107, E3 +171280.631}
SPL {X  -162.820, Y  +425.935, Z    +0.000, E1   +68.194, E3 +171295.687}
SPL {X  -162.820, Y  +409.792, Z    +0.000, E1   +68.121, E3 +171309.611}
SPL {X  -162.820, Y  +394.392, Z    +0.000, E1   +68.165, E3 +171322.185}
SPL {X  -162.820, Y  +385.264, Z    +0.000, E1   +67.766, E3 +171333.100}
ENDSPLINE

SPLINE
SPL {X  -162.820, Y  +401.104, Z    +0.000, E1   +65.023, E3 +171340.826}
ENDSPLINE

SPLINE
SPL {X  -162.820, Y  +386.513, Z    +0.000, E1   +65.423, E3 +171351.821}
SPL {X  -162.431, Y  +369.249, Z    +0.000, E1   +66.195, E3 +171361.823}
SPL {X  -160.017, Y  +350.416, Z    +0.000, E1   +67.091, E3 +171371.492}
SPL {X  -157.549, Y  +339.407, Z    +0.000, E1   +67.028, E3 +171381.368}
SPL {X  -154.848, Y  +330.175, Z    +0.000, E1   +66.891, E3 +171390.261}
SPL {X  -151.242, Y  +320.199, Z    +0.000, E1   +66.443, E3 +171402.062}
SPL {X  -147.540, Y  +311.636, Z    +0.000, E1   +65.718, E3 +171414.041}
SPL {X  -144.094, Y  +304.689, Z    +0.000, E1   +65.338, E3 +171422.255}
SPL {X  -141.093, Y  +299.241, Z    +0.000, E1   +65.039, E3 +171428.568}
SPL {X  -138.425, Y  +294.774, Z    +0.000, E1   +64.416, E3 +171435.752}
SPL {X  -135.581, Y  +290.344, Z    +0.000, E1   +63.996, E3 +171441.584}
SPL {X  -133.378, Y  +287.116, Z    +0.000, E1   +63.482, E3 +171446.748}
SPL {X  -128.896, Y  +281.020, Z    +0.000, E1   +64.005, E3 +171449.517}
SPL {X   -85.291, Y  +241.807, Z    +0.000, E1   +53.957, E3 +171594.925}
ENDSPLINE

SPLINE
SPL {X  -136.861, Y  +292.299, Z    +0.000, E1   +47.815, E3 +171722.546}
SPL {X  -156.420, Y  +335.300, Z    +0.000, E1   +31.885, E3 +171730.335}
SPL {X  -161.293, Y  +358.252, Z    +0.000, E1   +18.542, E3 +171732.053}
SPL {X  -162.487, Y  +370.094, Z    +0.000, E1   +10.144, E3 +171732.131}
SPL {X  -162.818, Y  +379.612, Z    +0.000, E1    +2.663, E3 +171732.106}
SPL {X  -162.820, Y  +382.500, Z    +0.000, E1    +0.000, E3 +171731.700}
SPL {X  -162.820, Y  +383.629, Z    +0.000, E1    -1.565, E3 +171731.393}
SPL {X  -162.820, Y  +386.448, Z    +0.000, E1    -6.246, E3 +171731.339}
SPL {X  -162.820, Y  +391.031, Z    +0.000, E1   -14.627, E3 +171731.397}
SPL {X  -162.820, Y  +397.383, Z    +0.000, E1   -27.100, E3 +171731.433}
SPL {X  -162.820, Y  +404.822, Z    +0.000, E1   -40.113, E3 +171731.084}
SPL {X  -162.820, Y  +416.103, Z    +0.000, E1   -54.033, E3 +171730.936}
SPL {X  -162.820, Y  +467.510, Z    +0.000, E1   -69.867, E3 +171744.514}
SPL {X  -162.820, Y  +604.717, Z    +0.000, E1   -70.047, E3 +171826.234}
SPL {X  -162.820, Y  +606.663, Z    +0.000, E1   -67.762, E3 +171847.282}
SPL {X  -162.820, Y  +626.641, Z    +0.000, E1   -67.759, E3 +171864.390}
SPL {X  -162.820, Y  +643.417, Z    +0.000, E1   -67.904, E3 +171877.206}
SPL {X  -162.820, Y  +654.663, Z    +0.000, E1   -67.744, E3 +171888.233}
SPL {X  -162.820, Y  +673.210, Z    +0.000, E1   -67.837, E3 +171903.266}
SPL {X  -162.071, Y  +689.103, Z    +0.000, E1   -67.763, E3 +171917.331}
SPL {X  -160.908, Y  +698.381, Z    +0.000, E1   -67.466, E3 +171927.570}
SPL {X  -158.503, Y  +710.744, Z    +0.000, E1   -67.284, E3 +171939.800}
SPL {X  -155.060, Y  +723.165, Z    +0.000, E1   -66.797, E3 +171953.976}
SPL {X  -152.159, Y  +731.448, Z    +0.000, E1   -66.356, E3 +171964.106}
SPL {X  -149.129, Y  +738.853, Z    +0.000, E1   -66.010, E3 +171972.804}
SPL {X  -146.076, Y  +745.418, Z    +0.000, E1   -65.453, E3 +171981.965}
SPL {X  -142.207, Y  +752.793, Z    +0.000, E1   -65.028, E3 +171990.814}
SPL {X  -139.223, Y  +757.923, Z    +0.000, E1   -64.359, E3 +171998.784}
SPL {X  -135.604, Y  +763.621, Z    +0.000, E1   -63.883, E3 +172006.152}
SPL {X  -131.007, Y  +770.183, Z    +0.000, E1   -63.497, E3 +172013.437}
SPL {X   -85.750, Y  +811.910, Z    +0.000, E1   -55.921, E3 +172117.390}
ENDSPLINE

SPLINE
SPL {X  -114.463, Y  +789.295, Z    +0.000, E1   -54.865, E3 +172286.657}
SPL {X  -149.148, Y  +738.810, Z    +0.000, E1   -41.467, E3 +172297.728}
SPL {X  -159.693, Y  +705.258, Z    +0.000, E1   -25.118, E3 +172300.368}
SPL {X  -162.196, Y  +687.741, Z    +0.000, E1   -13.310, E3 +172301.333}
SPL {X  -162.718, Y  +679.252, Z    +0.000, E1    -6.705, E3 +172301.670}
SPL {X  -162.820, Y  +671.587, Z    +0.000, E1    -0.252, E3 +172301.069}
SPL {X  -162.820, Y  +668.947, Z    +0.000, E1    +4.071, E3 +172300.682}
SPL {X  -162.820, Y  +664.754, Z    +0.000, E1   +11.697, E3 +172300.681}
SPL {X  -162.820, Y  +658.944, Z    +0.000, E1   +23.544, E3 +172300.849}
SPL {X  -162.820, Y  +653.429, Z    +0.000, E1   +34.521, E3 +172300.239}
SPL {X  -162.820, Y  +647.179, Z    +0.000, E1   +44.317, E3 +172300.456}
SPL {X  -162.820, Y  +635.494, Z    +0.000, E1   +57.613, E3 +172300.049}
SPL {X  -162.820, Y  +626.637, Z    +0.000, E1   +64.941, E3 +172298.765}
SPL {X  -162.820, Y  +572.535, Z    +0.000, E1   +70.270, E3 +172321.621}
SPL {X  -162.820, Y  +446.522, Z    +0.000, E1   +69.253, E3 +172405.445}
SPL {X  -162.820, Y  +440.686, Z    +0.000, E1   +68.127, E3 +172420.319}
SPL {X  -162.820, Y  +421.575, Z    +0.000, E1   +68.212, E3 +172435.383}
SPL {X  -162.820, Y  +409.792, Z    +0.000, E1   +68.121, E3 +172445.974}
SPL {X  -162.820, Y  +394.392, Z    +0.000, E1   +68.165, E3 +172458.549}
SPL {X  -162.820, Y  +385.264, Z    +0.000, E1   +67.766, E3 +172469.464}
ENDSPLINE

SPLINE
SPL {X  -162.820, Y  +401.104, Z    +0.000, E1   +65.023, E3 +172477.189}
ENDSPLINE

SPLINE
SPL {X  -162.820, Y  +386.513, Z    +0.000, E1   +65.423, E3 +172488.185}
SPL {X  -162.431, Y  +369.249, Z    +0.000, E1   +66.195, E3 +172498.186}
SPL {X  -160.017, Y  +350.416, Z    +0.000, E1   +67.091, E3 +172507.856}
SPL {X  -156.713, Y  +336.324, Z    +0.000, E1   +67.030, E3 +172520.452}
SPL {X  -153.279, Y  +325.584, Z    +0.000, E1   +66.662, E3 +172532.217}
SPL {X  -150.291, Y  +317.867, Z    +0.000, E1   +66.312, E3 +172541.136}
SPL {X  -147.540, Y  +311.636, Z    +0.000, E1   +65.718, E3 +172550.404}
SPL {X  -144.094, Y  +304.689, Z    +0.000, E1   +65.338, E3 +172558.619}
SPL {X  -141.093, Y  +299.241, Z    +0.000, E1   +65.039, E3 +172564.932}
SPL {X  -138.425, Y  +294.774, Z    +0.000, E1   +64.416, E3 +172572.116}
SPL {X  -134.374, Y  +288.555, Z    +0.000, E1   +63.758, E3 +172580.758}
SPL {X  -128.896, Y  +281.020, Z    +0.000, E1   +64.005, E3 +172585.881}
SPL {X   -85.291, Y  +241.807, Z    +0.000, E1   +53.957, E3 +172731.289}
ENDSPLINE

SPLINE
SPL {X  -136.861, Y  +292.299, Z    +0.000, E1   +47.815, E3 +172858.910}
SPL {X  -152.886, Y  +324.498, Z    +0.000, E1   +36.840, E3 +172865.591}
SPL {X  -158.256, Y  +342.219, Z    +0.000, E1   +28.198, E3 +172867.224}
SPL {X  -161.293, Y  +358.252, Z    +0.000, E1   +18.542, E3 +172868.416}
SPL {X  -162.687, Y  +373.932, Z    +0.000, E1    +7.306, E3 +172868.552}
SPL {X  -162.820, Y  +382.323, Z    +0.000, E1    +0.244, E3 +172868.111}
SPL {X  -162.820, Y  +383.629, Z    +0.000, E1    -1.565, E3 +172867.757}
SPL {X  -162.820, Y  +386.448, Z    +0.000, E1    -6.246, E3 +172867.702}
SPL {X  -162.820, Y  +391.031, Z    +0.000, E1   -14.627, E3 +172867.761}
SPL {X  -162.820, Y  +397.383, Z    +0.000, E1   -27.100, E3 +172867.796}
SPL {X  -162.820, Y  +404.822, Z    +0.000, E1   -40.113, E3 +172867.448}
SPL {X  -162.820, Y  +416.103, Z    +0.000, E1   -54.033, E3 +172867.300}
SPL {X  -162.820, Y  +472.592, Z    +0.000, E1   -70.190, E3 +172882.902}
SPL {X  -162.820, Y  +605.049, Z    +0.000, E1   -68.347, E3 +172977.384}
SPL {X  -162.820, Y  +616.480, Z    +0.000, E1   -67.752, E3 +172992.076}
SPL {X  -162.820, Y  +631.154, Z    +0.000, E1   -67.735, E3 +173004.611}
SPL {X  -162.820, Y  +647.590, Z    +0.000, E1   -67.861, E3 +173017.646}
SPL {X  -162.820, Y  +663.021, Z    +0.000, E1   -67.764, E3 +173031.484}
SPL {X  -162.799, Y  +676.123, Z    +0.000, E1   -67.801, E3 +173042.287}
SPL {X  -162.071, Y  +689.103, Z    +0.000, E1   -67.763, E3 +173053.694}
SPL {X  -160.908, Y  +698.381, Z    +0.000, E1   -67.466, E3 +173063.934}
SPL {X  -158.503, Y  +710.744, Z    +0.000, E1   -67.284, E3 +173076.163}
SPL {X  -155.060, Y  +723.165, Z    +0.000, E1   -66.797, E3 +173090.339}
SPL {X  -152.159, Y  +731.448, Z    +0.000, E1   -66.356, E3 +173100.470}
SPL {X  -149.129, Y  +738.853, Z    +0.000, E1   -66.010, E3 +173109.167}
SPL {X  -146.076, Y  +745.418, Z    +0.000, E1   -65.453, E3 +173118.329}
SPL {X  -143.238, Y  +750.916, Z    +0.000, E1   -65.112, E3 +173125.013}
SPL {X  -139.960, Y  +756.696, Z    +0.000, E1   -64.606, E3 +173132.914}
SPL {X  -136.860, Y  +761.702, Z    +0.000, E1   -64.057, E3 +173139.908}
SPL {X  -134.751, Y  +764.892, Z    +0.000, E1   -63.716, E3 +173144.303}
SPL {X  -131.007, Y  +770.183, Z    +0.000, E1   -63.497, E3 +173149.801}
SPL {X   -85.750, Y  +811.910, Z    +0.000, E1   -55.921, E3 +173253.754}
ENDSPLINE

SPLINE
SPL {X  -114.463, Y  +789.295, Z    +0.000, E1   -54.865, E3 +173423.021}
SPL {X  -144.553, Y  +748.431, Z    +0.000, E1   -44.979, E3 +173433.729}
SPL {X  -156.024, Y  +720.050, Z    +0.000, E1   -33.178, E3 +173435.295}
SPL {X  -160.714, Y  +699.606, Z    +0.000, E1   -21.520, E3 +173437.169}
SPL {X  -162.196, Y  +687.741, Z    +0.000, E1   -13.310, E3 +173437.697}
SPL {X  -162.791, Y  +676.596, Z    +0.000, E1    -4.586, E3 +173437.981}
SPL {X  -162.820, Y  +671.548, Z    +0.000, E1    -0.068, E3 +173437.458}
SPL {X  -162.820, Y  +669.949, Z    +0.000, E1    +2.213, E3 +173437.145}
SPL {X  -162.820, Y  +664.754, Z    +0.000, E1   +11.697, E3 +173437.044}
SPL {X  -162.820, Y  +658.944, Z    +0.000, E1   +23.544, E3 +173437.212}
SPL {X  -162.820, Y  +650.349, Z    +0.000, E1   +39.427, E3 +173436.710}
SPL {X  -162.820, Y  +635.494, Z    +0.000, E1   +57.613, E3 +173436.413}
SPL {X  -162.820, Y  +626.637, Z    +0.000, E1   +64.941, E3 +173435.128}
SPL {X  -162.820, Y  +572.535, Z    +0.000, E1   +70.270, E3 +173457.984}
SPL {X  -162.820, Y  +446.522, Z    +0.000, E1   +69.253, E3 +173541.808}
SPL {X  -162.820, Y  +440.686, Z    +0.000, E1   +68.127, E3 +173556.683}
SPL {X  -162.820, Y  +421.575, Z    +0.000, E1   +68.212, E3 +173571.747}
SPL {X  -162.820, Y  +409.792, Z    +0.000, E1   +68.121, E3 +173582.338}
SPL {X  -162.820, Y  +394.392, Z    +0.000, E1   +68.165, E3 +173594.912}
SPL {X  -162.820, Y  +385.264, Z    +0.000, E1   +67.766, E3 +173605.827}
ENDSPLINE

SPLINE
SPL {X  -162.820, Y  +401.104, Z    +0.000, E1   +65.023, E3 +173613.553}
ENDSPLINE

SPLINE
SPL {X  -162.820, Y  +386.513, Z    +0.000, E1   +65.423, E3 +173624.548}
SPL {X  -162.431, Y  +369.249, Z    +0.000, E1   +66.195, E3 +173634.550}
SPL {X  -160.017, Y  +350.416, Z    +0.000, E1   +67.091, E3 +173644.220}
SPL {X  -156.713, Y  +336.324, Z    +0.000, E1   +67.030, E3 +173656.816}
SPL {X  -153.279, Y  +325.584, Z    +0.000, E1   +66.662, E3 +173668.581}
SPL {X  -149.546, Y  +316.107, Z    +0.000, E1   +66.216, E3 +173679.757}
SPL {X  -147.033, Y  +310.560, Z    +0.000, E1   +65.497, E3 +173688.971}
SPL {X  -144.094, Y  +304.689, Z    +0.000, E1   +65.338, E3 +173694.983}
SPL {X  -141.093, Y  +299.241, Z    +0.000, E1   +65.039, E3 +173701.295}
SPL {X  -138.425, Y  +294.774, Z    +0.000, E1   +64.416, E3 +173708.479}
SPL {X  -134.374, Y  +288.555, Z    +0.000, E1   +63.758, E3 +173717.121}
SPL {X  -128.896, Y  +281.020, Z    +0.000, E1   +64.005, E3 +173722.244}
SPL {X   -85.291, Y  +241.807, Z    +0.000, E1   +53.957, E3 +173867.652}
ENDSPLINE

SPLINE
SPL {X  -136.861, Y  +292.299, Z    +0.000, E1   +47.815, E3 +173995.273}
SPL {X  -156.420, Y  +335.300, Z    +0.000, E1   +31.885, E3 +174003.062}
SPL {X  -161.293, Y  +358.252, Z    +0.000, E1   +18.542, E3 +174004.780}
SPL {X  -162.487, Y  +370.094, Z    +0.000, E1   +10.144, E3 +174004.858}
SPL {X  -162.818, Y  +379.612, Z    +0.000, E1    +2.663, E3 +174004.834}
SPL {X  -162.820, Y  +382.500, Z    +0.000, E1    +0.000, E3 +174004.427}
SPL {X  -162.820, Y  +383.629, Z    +0.000, E1    -1.565, E3 +174004.120}
SPL {X  -162.820, Y  +387.649, Z    +0.000, E1    -8.215, E3 +174004.108}
SPL {X  -162.820, Y  +392.460, Z    +0.000, E1   -17.627, E3 +174004.090}
SPL {X  -162.820, Y  +397.383, Z    +0.000, E1   -27.100, E3 +174004.160}
SPL {X  -162.820, Y  +404.822, Z    +0.000, E1   -40.113, E3 +174003.811}
SPL {X  -162.820, Y  +416.103, Z    +0.000, E1   -54.033, E3 +174003.663}
SPL {X  -162.820, Y  +472.592, Z    +0.000, E1   -70.190, E3 +174019.265}
SPL {X  -162.820, Y  +605.049, Z    +0.000, E1   -68.347, E3 +174113.747}
SPL {X  -162.820, Y  +616.480, Z    +0.000, E1   -67.752, E3 +174128.440}
SPL {X  -162.820, Y  +631.154, Z    +0.000, E1   -67.735, E3 +174140.975}
SPL {X  -162.820, Y  +647.590, Z    +0.000, E1   -67.861, E3 +174154.010}
SPL {X  -162.820, Y  +663.021, Z    +0.000, E1   -67.764, E3 +174167.847}
SPL {X  -162.642, Y  +681.112, Z    +0.000, E1   -67.812, E3 +174182.999}
SPL {X  -161.154, Y  +696.734, Z    +0.000, E1   -67.591, E3 +174197.996}
SPL {X  -158.503, Y  +710.744, Z    +0.000, E1   -67.284, E3 +174212.527}
SPL {X  -155.060, Y  +723.165, Z    +0.000, E1   -66.797, E3 +174226.703}
SPL {X  -151.511, Y  +733.123, Z    +0.000, E1   -66.286, E3 +174238.857}
SPL {X  -147.735, Y  +741.944, Z    +0.000, E1   -65.827, E3 +174249.383}
SPL {X  -144.196, Y  +749.116, Z    +0.000, E1   -65.203, E3 +174259.383}
SPL {X  -139.960, Y  +756.696, Z    +0.000, E1   -64.606, E3 +174269.277}
SPL {X  -135.604, Y  +763.621, Z    +0.000, E1   -63.883, E3 +174278.879}
SPL {X  -131.007, Y  +770.183, Z    +0.000, E1   -63.497, E3 +174286.165}
SPL {X   -85.750, Y  +811.910, Z    +0.000, E1   -55.921, E3 +174390.117}
ENDSPLINE

SPLINE
SPL {X  -114.463, Y  +789.295, Z    +0.000, E1   -54.865, E3 +174559.384}
SPL {X  -149.148, Y  +738.810, Z    +0.000, E1   -41.467, E3 +174570.455}
SPL {X  -159.693, Y  +705.258, Z    +0.000, E1   -25.118, E3 +174573.095}
SPL {X  -162.196, Y  +687.741, Z    +0.000, E1   -13.310, E3 +174574.060}
SPL {X  -162.791, Y  +676.596, Z    +0.000, E1    -4.586, E3 +174574.344}
SPL {X  -162.820, Y  +671.548, Z    +0.000, E1    -0.068, E3 +174573.821}
SPL {X  -162.820, Y  +669.949, Z    +0.000, E1    +2.213, E3 +174573.509}
SPL {X  -162.820, Y  +664.754, Z    +0.000, E1   +11.697, E3 +174573.408}
SPL {X  -162.820, Y  +658.944, Z    +0.000, E1   +23.544, E3 +174573.576}
SPL {X  -162.820, Y  +653.429, Z    +0.000, E1   +34.521, E3 +174572.967}
SPL {X  -162.820, Y  +647.179, Z    +0.000, E1   +44.317, E3 +174573.183}
SPL {X  -162.820, Y  +632.228, Z    +0.000, E1   +60.508, E3 +174572.303}
SPL {X  -162.820, Y  +572.535, Z    +0.000, E1   +70.270, E3 +174594.348}
SPL {X  -162.820, Y  +446.522, Z    +0.000, E1   +69.253, E3 +174678.172}
SPL {X  -162.820, Y  +444.665, Z    +0.000, E1   +68.107, E3 +174689.722}
SPL {X  -162.820, Y  +425.935, Z    +0.000, E1   +68.194, E3 +174704.778}
SPL {X  -162.820, Y  +405.187, Z    +0.000, E1   +68.161, E3 +174722.366}
SPL {X  -162.820, Y  +387.680, Z    +0.000, E1   +67.977, E3 +174738.555}
ENDSPLINE

SPLINE
SPL {X  -162.820, Y  +397.358, Z    +0.000, E1   +65.083, E3 +174753.193}
ENDSPLINE

SPLINE
SPL {X  -162.719, Y  +374.774, Z    +0.000, E1   +65.968, E3 +174767.677}
SPL {X  -160.017, Y  +350.416, Z    +0.000, E1   +67.091, E3 +174780.583}
SPL {X  -156.713, Y  +336.324, Z    +0.000, E1   +67.030, E3 +174793.180}
SPL {X  -153.279, Y  +325.584, Z    +0.000, E1   +66.662, E3 +174804.945}
SPL {X  -150.291, Y  +317.867, Z    +0.000, E1   +66.312, E3 +174813.864}
SPL {X  -147.540, Y  +311.636, Z    +0.000, E1   +65.718, E3 +174823.132}
SPL {X  -144.094, Y  +304.689, Z    +0.000, E1   +65.338, E3 +174831.346}
SPL {X  -141.093, Y  +299.241, Z    +0.000, E1   +65.039, E3 +174837.659}
SPL {X  -138.425, Y  +294.774, Z    +0.000, E1   +64.416, E3 +174844.843}
SPL {X  -134.374, Y  +288.555, Z    +0.000, E1   +63.758, E3 +174853.485}
SPL {X  -128.896, Y  +281.020, Z    +0.000, E1   +64.005, E3 +174858.608}
SPL {X   -85.291, Y  +241.807, Z    +0.000, E1   +53.957, E3 +175004.016}
ENDSPLINE

SPLINE
SPL {X  -136.861, Y  +292.299, Z    +0.000, E1   +47.815, E3 +175131.637}
SPL {X  -156.420, Y  +335.300, Z    +0.000, E1   +31.885, E3 +175139.426}
SPL {X  -161.293, Y  +358.252, Z    +0.000, E1   +18.542, E3 +175141.144}
SPL {X  -162.687, Y  +373.932, Z    +0.000, E1    +7.306, E3 +175141.279}
SPL {X  -162.820, Y  +382.323, Z    +0.000, E1    +0.244, E3 +175140.838}
SPL {X  -162.820, Y  +383.629, Z    +0.000, E1    -1.565, E3 +175140.484}
SPL {X  -162.820, Y  +386.448, Z    +0.000, E1    -6.246, E3 +175140.429}
SPL {X  -162.820, Y  +391.031, Z    +0.000, E1   -14.627, E3 +175140.488}
SPL {X  -162.820, Y  +397.383, Z    +0.000, E1   -27.100, E3 +175140.523}
SPL {X  -162.820, Y  +404.822, Z    +0.000, E1   -40.113, E3 +175140.175}
SPL {X  -162.820, Y  +416.103, Z    +0.000, E1   -54.033, E3 +175140.027}
SPL {X  -162.820, Y  +472.592, Z    +0.000, E1   -70.190, E3 +175155.629}
SPL {X  -162.820, Y  +611.623, Z    +0.000, E1   -69.722, E3 +175242.962}
ENDSPLINE

SPLINE
SPL {X  -162.820, Y  +606.663, Z    +0.000, E1   -67.762, E3 +175256.373}
ENDSPLINE

SPLINE
SPL {X  -162.820, Y  +626.641, Z    +0.000, E1   -67.759, E3 +175273.480}
SPL {X  -162.820, Y  +643.417, Z    +0.000, E1   -67.904, E3 +175286.297}
SPL {X  -162.820, Y  +654.663, Z    +0.000, E1   -67.744, E3 +175297.323}
SPL {X  -162.820, Y  +673.210, Z    +0.000, E1   -67.837, E3 +175312.357}
SPL {X  -162.071, Y  +689.103, Z    +0.000, E1   -67.763, E3 +175326.422}
SPL {X  -160.908, Y  +698.381, Z    +0.000, E1   -67.466, E3 +175336.661}
SPL {X  -158.503, Y  +710.744, Z    +0.000, E1   -67.284, E3 +175348.891}
SPL {X  -155.060, Y  +723.165, Z    +0.000, E1   -66.797, E3 +175363.067}
SPL {X  -152.159, Y  +731.448, Z    +0.000, E1   -66.356, E3 +175373.197}
SPL {X  -149.129, Y  +738.853, Z    +0.000, E1   -66.010, E3 +175381.895}
SPL {X  -146.076, Y  +745.418, Z    +0.000, E1   -65.453, E3 +175391.056}
SPL {X  -143.238, Y  +750.916, Z    +0.000, E1   -65.112, E3 +175397.741}
SPL {X  -139.960, Y  +756.696, Z    +0.000, E1   -64.606, E3 +175405.641}
SPL {X  -135.604, Y  +763.621, Z    +0.000, E1   -63.883, E3 +175415.243}
SPL {X  -131.007, Y  +770.183, Z    +0.000, E1   -63.497, E3 +175422.528}
SPL {X   -85.750, Y  +811.910, Z    +0.000, E1   -55.921, E3 +175526.481}
ENDSPLINE

SPLINE
SPL {X  -114.463, Y  +789.295, Z    +0.000, E1   -54.865, E3 +175695.748}
SPL {X  -149.148, Y  +738.810, Z    +0.000, E1   -41.467, E3 +175706.819}
SPL {X  -159.693, Y  +705.258, Z    +0.000, E1   -25.118, E3 +175709.459}
SPL {X  -162.196, Y  +687.741, Z    +0.000, E1   -13.310, E3 +175710.424}
SPL {X  -162.718, Y  +679.252, Z    +0.000, E1    -6.705, E3 +175710.761}
SPL {X  -162.820, Y  +671.587, Z    +0.000, E1    -0.252, E3 +175710.160}
SPL {X  -162.820, Y  +667.797, Z    +0.000, E1    +5.943, E3 +175709.784}
SPL {X  -162.820, Y  +663.306, Z    +0.000, E1   +14.820, E3 +175709.751}
SPL {X  -162.820, Y  +658.944, Z    +0.000, E1   +23.544, E3 +175709.940}
SPL {X  -162.820, Y  +650.349, Z    +0.000, E1   +39.427, E3 +175709.437}
SPL {X  -162.820, Y  +632.228, Z    +0.000, E1   +60.508, E3 +175708.667}
SPL {X  -162.820, Y  +572.535, Z    +0.000, E1   +70.270, E3 +175730.712}
SPL {X  -162.820, Y  +446.522, Z    +0.000, E1   +69.253, E3 +175814.536}
SPL {X  -162.820, Y  +440.686, Z    +0.000, E1   +68.127, E3 +175829.410}
SPL {X  -162.820, Y  +421.575, Z    +0.000, E1   +68.212, E3 +175844.474}
SPL {X  -162.820, Y  +409.792, Z    +0.000, E1   +68.121, E3 +175855.065}
SPL {X  -162.820, Y  +394.392, Z    +0.000, E1   +68.165, E3 +175867.639}
SPL {X  -162.820, Y  +385.264, Z    +0.000, E1   +67.766, E3 +175878.555}
ENDSPLINE

SPLINE
SPL {X  -162.820, Y  +397.358, Z    +0.000, E1   +65.083, E3 +175889.557}
ENDSPLINE

SPLINE
SPL {X  -162.719, Y  +374.774, Z    +0.000, E1   +65.968, E3 +175904.041}
SPL {X  -161.214, Y  +357.685, Z    +0.000, E1   +66.686, E3 +175913.796}
SPL {X  -158.043, Y  +341.350, Z    +0.000, E1   +67.216, E3 +175923.904}
SPL {X  -154.848, Y  +330.175, Z    +0.000, E1   +66.891, E3 +175935.716}
SPL {X  -152.657, Y  +323.878, Z    +0.000, E1   +66.551, E3 +175943.450}
SPL {X  -149.546, Y  +316.107, Z    +0.000, E1   +66.216, E3 +175952.484}
SPL {X  -147.033, Y  +310.560, Z    +0.000, E1   +65.497, E3 +175961.698}
SPL {X  -144.094, Y  +304.689, Z    +0.000, E1   +65.338, E3 +175967.710}
SPL {X  -141.093, Y  +299.241, Z    +0.000, E1   +65.039, E3 +175974.023}
SPL {X  -138.425, Y  +294.774, Z    +0.000, E1   +64.416, E3 +175981.207}
SPL {X  -135.581, Y  +290.344, Z    +0.000, E1   +63.996, E3 +175987.039}
SPL {X  -133.378, Y  +287.116, Z    +0.000, E1   +63.482, E3 +175992.203}
SPL {X  -128.896, Y  +281.020, Z    +0.000, E1   +64.005, E3 +175994.972}
SPL {X   -85.291, Y  +241.807, Z    +0.000, E1   +53.957, E3 +176140.380}
ENDSPLINE

SPLINE
SPL {X  -136.861, Y  +292.299, Z    +0.000, E1   +47.815, E3 +176268.001}
SPL {X  -156.420, Y  +335.300, Z    +0.000, E1   +31.885, E3 +176275.790}
SPL {X  -161.293, Y  +358.252, Z    +0.000, E1   +18.542, E3 +176277.507}
SPL {X  -162.487, Y  +370.094, Z    +0.000, E1   +10.144, E3 +176277.585}
SPL {X  -162.818, Y  +379.612, Z    +0.000, E1    +2.663, E3 +176277.561}
SPL {X  -162.820, Y  +382.500, Z    +0.000, E1    +0.000, E3 +176277.154}
SPL {X  -162.820, Y  +383.629, Z    +0.000, E1    -1.565, E3 +176276.848}
SPL {X  -162.820, Y  +387.649, Z    +0.000, E1    -8.215, E3 +176276.836}
SPL {X  -162.820, Y  +392.460, Z    +0.000, E1   -17.627, E3 +176276.817}
SPL {X  -162.820, Y  +397.383, Z    +0.000, E1   -27.100, E3 +176276.887}
SPL {X  -162.820, Y  +404.822, Z    +0.000, E1   -40.113, E3 +176276.539}
SPL {X  -162.820, Y  +416.103, Z    +0.000, E1   -54.033, E3 +176276.391}
SPL {X  -162.820, Y  +472.592, Z    +0.000, E1   -70.190, E3 +176291.993}
SPL {X  -162.820, Y  +605.049, Z    +0.000, E1   -68.347, E3 +176386.474}
SPL {X  -162.820, Y  +616.480, Z    +0.000, E1   -67.752, E3 +176401.167}
SPL {X  -162.820, Y  +631.154, Z    +0.000, E1   -67.735, E3 +176413.702}
SPL {X  -162.820, Y  +647.590, Z    +0.000, E1   -67.861, E3 +176426.737}
SPL {X  -162.820, Y  +663.021, Z    +0.000, E1   -67.764, E3 +176440.575}
SPL {X  -162.642, Y  +681.112, Z    +0.000, E1   -67.812, E3 +176455.726}
SPL {X  -161.154, Y  +696.734, Z    +0.000, E1   -67.591, E3 +176470.723}
SPL {X  -158.503, Y  +710.744, Z    +0.000, E1   -67.284, E3 +176485.254}
SPL {X  -155.060, Y  +723.165, Z    +0.000, E1   -66.797, E3 +176499.430}
SPL {X  -151.511, Y  +733.123, Z    +0.000, E1   -66.286, E3 +176511.584}
SPL {X  -147.735, Y  +741.944, Z    +0.000, E1   -65.827, E3 +176522.110}
SPL {X  -144.196, Y  +749.116, Z    +0.000, E1   -65.203, E3 +176532.111}
SPL {X  -139.960, Y  +756.696, Z    +0.000, E1   -64.606, E3 +176542.005}
SPL {X  -135.604, Y  +763.621, Z    +0.000, E1   -63.883, E3 +176551.607}
SPL {X  -131.007, Y  +770.183, Z    +0.000, E1   -63.497, E3 +176558.892}
SPL {X   -85.750, Y  +811.910, Z    +0.000, E1   -55.921, E3 +176662.844}
ENDSPLINE

SPLINE
SPL {X  -114.463, Y  +789.295, Z    +0.000, E1   -54.865, E3 +176832.111}
SPL {X  -149.148, Y  +738.810, Z    +0.000, E1   -41.467, E3 +176843.183}
SPL {X  -159.693, Y  +705.258, Z    +0.000, E1   -25.118, E3 +176845.822}
SPL {X  -162.196, Y  +687.741, Z    +0.000, E1   -13.310, E3 +176846.787}
SPL {X  -162.791, Y  +676.596, Z    +0.000, E1    -4.586, E3 +176847.072}
SPL {X  -162.820, Y  +671.548, Z    +0.000, E1    -0.068, E3 +176846.549}
SPL {X  -162.820, Y  +669.949, Z    +0.000, E1    +2.213, E3 +176846.236}
SPL {X  -162.820, Y  +664.754, Z    +0.000, E1   +11.697, E3 +176846.135}
SPL {X  -162.820, Y  +658.944, Z    +0.000, E1   +23.544, E3 +176846.303}
SPL {X  -162.820, Y  +653.429, Z    +0.000, E1   +34.521, E3 +176845.694}
SPL {X  -162.820, Y  +647.179, Z    +0.000, E1   +44.317, E3 +176845.910}
SPL {X  -162.820, Y  +632.228, Z    +0.000, E1   +60.508, E3 +176845.031}
SPL {X  -162.820, Y  +572.535, Z    +0.000, E1   +70.270, E3 +176867.075}
SPL {X  -162.820, Y  +446.522, Z    +0.000, E1   +69.253, E3 +176950.899}
SPL {X  -162.820, Y  +444.665, Z    +0.000, E1   +68.107, E3 +176962.449}
SPL {X  -162.820, Y  +425.935, Z    +0.000, E1   +68.194, E3 +176977.505}
SPL {X  -162.820, Y  +405.187, Z    +0.000, E1   +68.161, E3 +176995.094}
SPL {X  -162.820, Y  +387.680, Z    +0.000, E1   +67.977, E3 +177011.282}
ENDSPLINE

SPLINE
SPL {X  -162.820, Y  +397.358, Z    +0.000, E1   +65.083, E3 +177025.920}
ENDSPLINE

SPLINE
SPL {X  -162.719, Y  +374.774, Z    +0.000, E1   +65.968, E3 +177040.405}
SPL {X  -160.034, Y  +350.509, Z    +0.000, E1   +67.062, E3 +177053.479}
SPL {X  -158.976, Y  +345.331, Z    +0.000, E1   +65.735, E3 +177068.474}
SPL {X  -155.590, Y  +332.521, Z    +0.000, E1   +65.288, E3 +177083.525}
SPL {X  -151.631, Y  +321.184, Z    +0.000, E1   +64.776, E3 +177097.378}
SPL {X  -147.832, Y  +312.265, Z    +0.000, E1   +64.201, E3 +177109.188}
SPL {X  -145.264, Y  +306.955, Z    +0.000, E1   +63.555, E3 +177117.794}
SPL {X  -142.454, Y  +301.650, Z    +0.000, E1   +63.360, E3 +177123.798}
SPL {X  -139.696, Y  +296.861, Z    +0.000, E1   +62.910, E3 +177130.565}
SPL {X  -137.330, Y  +293.030, Z    +0.000, E1   +62.290, E3 +177137.190}
SPL {X  -134.245, Y  +288.366, Z    +0.000, E1   +62.031, E3 +177142.672}
SPL {X  -128.642, Y  +280.693, Z    +0.000, E1   +63.351, E3 +177143.665}
SPL {X   -90.696, Y  +245.280, Z    +0.000, E1   +54.124, E3 +177264.354}
ENDSPLINE

